(* CoDeSys 2.3.9.59 project: wago_881.pro *)
(* Libraries: WagoLibEthernet_01.lib*10.7.18 06:47:36, SysLibSockets.lib 10.2.11 08:20:54, DALI_02_v2.12.lib*17.1.19 11:19:38, WagoLibReset.lib 2.12.10 13:48:32, SysLibFile.lib 2.12.10 13:48:34, DMXStageProfi_01.lib*19.6.19 09:17:07, Visual.lib 2.12.10 13:48:34, mod_com.lib 2.12.10 13:48:32, Ethernet.lib 2.12.10 13:48:32, SysLibGetAddress.lib 2.12.10 13:48:32, SysLibTime.lib 2.12.10 13:48:32, Standard.lib 2.12.10 13:48:34, SYSLIBCALLBACK.LIB 2.12.10 13:48:32 *)

(* PLC configuration (modules and I/O channels)
K-Bus [K_Bus] node 0, in %IB0 out %QB0
Fieldbus variables [FB_VARS] node 1, in %IB512 out %QB512
*)

(* Task configuration *)
TASK MainTask (PRIORITY := 1); (* freewheeling *)
	PLC_PRG();
END_TASK
TASK DMXTask (PRIORITY := 2, INTERVAL := T#10ms);
	DMX();
END_TASK

(* Global variable list: Variables_Globales *)
VAR_GLOBAL
	ConfigDone: BOOL := FALSE; (* Do the config only one time *)
	info : ARRAY[0..63] OF MODULE_INFO; (* I/O Module infos *)

	LedMode: BYTE := 0;

	(* modules infos *)
	nb_module: BYTE;
	nb_module_in: BYTE;
	nb_module_out: BYTE;
	nb_module_analog_in: BYTE;
	nb_module_analog_out: BYTE;
	start_addr_in: WORD;
	start_addr_out: WORD;
	nb_input_digital: WORD;
	nb_output_digital: WORD;

	(* All inputs events *)
	event: ARRAY[0..512] OF INTER_EVENT; (* See Rules mapping below *)
	lights: ARRAY[0..63] OF BYTE;	(* MAX of 256/8 = 32 digital output modules as lights *)
									(* We store only the boolean state of each light *)
	volets: ARRAY[0..512] OF VOLET; (* MAX of 256/8 = 32 digital output modules as volets *)

	HEARTBEAT: BOOL := FALSE;

	OutArrState: ARRAY[0..512] OF BYTE;	(* state of outputs *)

	impulse_time: TIME := T#300ms;

	(* DALI *)
	DALIJoblist: FbDALI_Joblist;

	Dali_switch: FbDALI_SwitchValue;
	DALIDimmValue: FbDALI_StatusDimmValue;

	(*
		Modbus addresses mapping:
			- [4096..4352] : Standard digital outputs
			- [6144..6244] : KNX inputs/outputs
	*)

	netOutStandard AT %IB512: ARRAY[0..31] OF BYTE;

	netOutKNX AT %IB768: ARRAY[0..12] OF BYTE;
	netInKNX AT %QB768: ARRAY[0..12] OF BYTE;

	write_word: WRITE_OUTPUT_WORD;
	write_bit: WRITE_OUTPUT_BIT;
	read_bit: READ_INPUT_BIT;

END_VAR
VAR_GLOBAL RETAIN
	(* Rules mapping:
		- [0..256] : standard digital inputs
		- [257..357]: knx digital inputs
	*)
	output_type: ARRAY[0..512] OF OUTPUT_TYPE; (* The type of each output *)
	output_addr: ARRAY[0..512] OF OUTPUT_ADDR; (* The addresses for each type *)

    volets_position: ARRAY[0..100] OF DWORD;

	(* DMX Values *)
	abDMX_Values: ARRAY [1..255] OF BYTE;
END_VAR

(* Data type *)
TYPE OUTPUT_ADDR :
STRUCT

	(* the first ouput address, only needed *)
	ADDR1: WORD;
	(* the second address used only for the VOLET function bloc *)
	ADDR2: WORD;

	(* If SameAs <> -1, then a input is wired the same as the specified ID *)
	SameAs: INT := -1;

END_STRUCT
END_TYPE

(* Data type *)
(* Enumerate all type of output.
	NONE: Do nothing.
	TELERUPTEUR: Simulate a telerupteur.
	DIRECT: The input is directly "wired" to the output.
	VOLET: Simulate a volet with one button and 2 output (up and down).
	TELERUPTEUR_DALI: Controls a DALI lamp
	TELERUPTEUR_DALI_GROUP: Controls a DALI group
	KNX_OUTPUT: Simulate a telerupteur with a KNX bool output
*)

TYPE OUTPUT_TYPE : (NONE,
					TELERUPTEUR, DIRECT,
					VOLET, VOLET_IMPULSE,
					TELERUPTEUR_DALI,
					TELERUPTEUR_DALI_GROUP,
					TELERUPTEUR_KNX_OUTPUT,
					DIRECT_KNX_OUTPUT);
END_TYPE

(* Data type *)
TYPE typEthernet_BUFFER :
	STRUCT
		Index		:	INT;
		Data		:	ARRAY[1..1500] OF BYTE;
	END_STRUCT
END_TYPE

(* Data type *)
(* Enumerate all type of output.
	NONE: Do nothing.
	TELERUPTEUR: Simulate a telerupteur.
	DIRECT: The input is directly "wired" to the output.
	VOLET: Simulate a volet with one button and 2 output (up and down).
*)

TYPE VOLET_MODE : (VOLET_STOP, VOLET_UP, VOLET_DOWN, IMP_UP, IMP_DOWN, IMP_STOP);
END_TYPE

(* POU PLC_PRG, ST *)
PROGRAM PLC_PRG
VAR
	i: INT;
	j: INT;
	start: BYTE;
	init_dali: BOOL := FALSE;
	valw: WORD;
	led: LedUsr;
END_VAR
(* Main PRG *)
Config_File_XML();

led(Mode := LedMode);

(* Start the config program *)
Config;

IF (Config.CONFIG_DALI = TRUE) THEN

	(* Call DALI jobs to send commands on the DALI bus *)
	DALIJoblist();
	DALI_Config();

	IF (init_dali = FALSE) THEN
		Dali_switch(xButton := FALSE);
		Dali_switch(bAddress := 255, xGroup := FALSE, bDimmLevel := 0,
				         xButton := TRUE);

		init_dali := TRUE;
	END_IF

END_IF

(* Read inputs and send their status on the network if they changed *)
SendInput;

(* Read a command from UDP *)
UDPServer;

IF (HEARTBEAT = FALSE) THEN
 	ManageOutput;
END_IF

IF (HEARTBEAT = FALSE) THEN

	j := start_addr_out / 8;
	FOR i := start_addr_out / 16 TO 15 DO
		valw := OutArrState[j + 1];
		write_word(WORD_ADDRESS := i, VALUE := SHL(valw, 8) + OutArrState[j]);
		j := j + 2;
	END_FOR
ELSE

	j := 0;
	FOR i := 0 TO 14 DO
		valw := netOutStandard[j + 1];
		write_word(WORD_ADDRESS := i + start_addr_out / 16, VALUE := SHL(valw, 8) + netOutStandard[j]);
		j := j + 2;
		OutArrState[j] := netOutStandard[j];
		OutArrState[j + 1] := netOutStandard[j + 1];
	END_FOR

END_IF
END_PROGRAM

(* POU LedUsr, ST *)
FUNCTION_BLOCK LedUsr
VAR_INPUT
	Mode: BYTE;

END_VAR
VAR_OUTPUT
END_VAR
VAR
	Sequence: ARRAY [0..4] OF FLASHING_SEQUENCE;
	ptrFS: POINTER TO FLASHING_SEQUENCE;

	i: BYTE := 0;
END_VAR
CASE Mode OF
	0 : i := 0;
	1 : i := 11; (* Mode Wago *)
	2 : i := 12; (* Mode PC *)
	3 : i := 13; (* Error *)
END_CASE

LedMode := 255;

CASE i OF
	0 : (* Init *)
		Sequence[0].Colour := ORANGE;
		Sequence[0].Frequency := 10;
		Sequence[0].Relation := 128;
		Sequence[0].Duration := t#0s;

		Sequence[1].Colour := ORANGE;
		Sequence[1].Frequency := 0;
		Sequence[1].Relation := 128;
		Sequence[1].Duration := t#0s;

		Sequence[2].Colour := GREEN;
		Sequence[2].Frequency := 0;
		Sequence[2].Relation := 128;
		Sequence[2].Duration := t#0s;

		Sequence[3].Colour := RED;
		Sequence[3].Frequency := 0;
		Sequence[3].Relation := 128;
		Sequence[3].Duration := t#0s;

		Sequence[4].Colour := ORANGE;
		Sequence[4].Frequency := 0;
		Sequence[4].Relation := 0;
		Sequence[4].Duration := t#0s;

		ptrFS := ADR(Sequence);
		SET_FLASHING_SEQUENCE(TRUE, ADR(ptrFS));

		i := 10;

	10: (* Start *)
		SET_FLASHING_SEQUENCE_INDEX(TRUE, TRUE, 0);
		START_FLASHING_SEQUENCE(TRUE);

		i := 255;

	11: (* Led Mode wago *)
		SET_FLASHING_SEQUENCE_INDEX(TRUE, TRUE, 1);

		i := 255;

	12: (* Led Mode PC *)
		SET_FLASHING_SEQUENCE_INDEX(TRUE, TRUE, 2);

		i := 255;

	13: (* Led Error *)
		SET_FLASHING_SEQUENCE_INDEX(TRUE, TRUE, 3);

		i := 255;

END_CASE
END_FUNCTION_BLOCK

(* POU Config_File_XML, ST *)
PROGRAM Config_File_XML
VAR RETAIN
	wModuleCount : WORD;
END_VAR
VAR CONSTANT
	STRING_1: STRING := '<?xml version="1.0" encoding="ISO-8859-1"?>$r$n';
	STRING_2: STRING := '<?xml-stylesheet type="text/xsl" href="/webserv/cplcfg/EA-config.xsl" ?>$R$n';
	STRING_3: STRING := '<WAGO>$R$n';
	STRING_4: STRING := '<Module ARTIKELNR="" MAP="PLC" LOC="ALL"></Module>$R$n';
	STRING_5: STRING := '</WAGO>$r$n';
END_VAR
VAR
	info : ARRAY[0..63] OF MODULE_INFO;
	access: MODULE_INFO_ACCESS;
	i: INT := 0;
	Status: BYTE := 0;
	DetectedModules: INT;
	FileHandle: DWORD;
	dwWrite: DWORD;
	NumberOfEntries: BYTE := 0;
	FileIsClosed: BOOL;
END_VAR
CASE Status OF
	0 :	ADD_PI_INFORMATION(EN:=TRUE, pAccess:=ADR(access), pInfo:=ADR(info));
		i:=0;
		WHILE info[i].physicalPos<>0
			DO
			i:=i+1;
		END_WHILE
		DetectedModules := i;
		Status := Status +1;
	1 :	IF DetectedModules = wModuleCount
			THEN
			Status := 255; (* Done *)
		ELSE
			Status := 10;
		END_IF
	10:	FileHandle:=SysFileOpen(FileName:='\etc\EA-config.xml', Mode:='w');
		IF FileHandle <> 0 THEN
			Status := Status+1;
		END_IF
	11:	dwWrite:=SysFileWrite(File:=FileHandle, Buffer:=ADR(STRING_1), Size:=LEN(STRING_1));
		IF dwWrite=LEN(STRING_1) THEN
			Status := Status+1;
		END_IF
	12:	dwWrite:=SysFileWrite(File:=FileHandle, Buffer:=ADR(STRING_2), Size:=LEN(STRING_2));
		IF dwWrite=LEN(STRING_2) THEN
			Status := Status+1;
		END_IF
	13:	dwWrite:=SysFileWrite(File:=FileHandle, Buffer:=ADR(STRING_3), Size:=LEN(STRING_3));
		IF dwWrite=LEN(STRING_3) THEN
			Status := Status+1;
		END_IF
	14:	dwWrite:=SysFileWrite(File:=FileHandle, Buffer:=ADR(STRING_4), Size:=LEN(STRING_4));
		IF dwWrite=LEN(STRING_4) THEN
			Status := Status+1;
			NumberOfEntries := NumberOfEntries+1;
		END_IF
	15: IF NumberOfEntries < DetectedModules
			THEN
			Status := Status -1;
		ELSE
			Status := Status +1;
		END_IF
	16:	dwWrite:=SysFileWrite(File:=FileHandle, Buffer:=ADR(STRING_5), Size:=LEN(STRING_5));
		IF dwWrite=LEN(STRING_5) THEN
			Status := Status+1;
		END_IF
	17:	FileIsClosed := SysFileClose(File:= FileHandle);
		IF FileIsClosed
			THEN
			Status := 20;
		END_IF
	20:	wModuleCount := DetectedModules;
		FirmwareReset(EN := TRUE);
END_CASE
END_PROGRAM

(* POU Config, ST *)
PROGRAM Config
VAR
	access : MODULE_INFO_ACCESS;
	cpt: BYTE;
	ethernet_config : ETHERNET_SET_VARIABLES;
	CONFIG_DALI: BOOL;
	first_in: BOOL := FALSE;
	first_out: BOOL := FALSE;
END_VAR
VAR_INPUT RETAIN
	SERVER_IP: DWORD;
	DALI_MODE: BYTE;
END_VAR
VAR CONSTANT
	CALAOS_VERSION_H: WORD := 2;
	CALAOS_VERSION_L: WORD := 3;
	DALI: BYTE := 1;
	DSI: BYTE := 2;
END_VAR
(* Do all the config job *)

IF (ConfigDone = FALSE) THEN

(* Get the module I/O Config *)
access.physicalPosTo := 0;
access.moduleType := 0;
ADD_PI_INFORMATION( 1, ADR(access), ADR(info[0]) );

FOR cpt := 0 TO 63 DO
	IF (info[cpt].moduleType = 0 AND info[cpt].physicalPos = 0) THEN
		cpt := 63; (* the end *)
	ELSE
		IF (info[cpt].moduleType = 641) THEN
			(* This is a DALI module *)
			CONFIG_DALI := TRUE;
		END_IF

		nb_module := nb_module + 1;
		IF ((info[cpt].desc.sizePAE > 8) AND (info[cpt].desc.channels > 0)) THEN
			nb_module_analog_in := nb_module_analog_in + 1;
(*			start_addr_in := start_addr_in + info[cpt].desc.sizePAE; *)
		END_IF
		IF ((info[cpt].desc.sizePAA > 8) AND (info[cpt].desc.channels > 0)) THEN
			nb_module_analog_out := nb_module_analog_out + 1;
(*			start_addr_out := start_addr_out + info[cpt].desc.sizePAA; *)
		END_IF
		IF ((info[cpt].desc.sizePAE <= 16) AND (info[cpt].desc.sizePAE > 0) AND (info[cpt].desc.channels = 0)) THEN
			nb_module_in := nb_module_in + 1;
			nb_input_digital := nb_input_digital + info[cpt].desc.sizePAE;

			IF (first_in = FALSE) THEN
				first_in := TRUE;
				start_addr_in := info[cpt].desc.posPAE;
			END_IF
		END_IF
		IF ((info[cpt].desc.sizePAA <= 16) AND (info[cpt].desc.sizePAA > 0) AND (info[cpt].desc.channels = 0)) THEN
			nb_module_out := nb_module_out + 1;
			nb_output_digital := nb_output_digital + info[cpt].desc.sizePAA;

			IF (first_out = FALSE) THEN
				first_out := TRUE;
				start_addr_out := info[cpt].desc.posPAA;
			END_IF
		END_IF

	END_IF
END_FOR

(* Start the heartbeat timer *)
(*HEARTBEAT_TIMER(IN:=FALSE, PT:=T#30s);*)
(*HEARTBEAT_TIMER(IN:=TRUE, PT:=T#30s);*)

(* Config du timout des sockets *)
ethernet_config(EN:=TRUE, BootpRequest:=0, ConnectionWdTime:=65535);

ConfigDone := TRUE;

END_IF
END_PROGRAM

(* POU SendInput, ST *)
PROGRAM SendInput
VAR
	cpt: INT;

	eth: Ethernet_Client;
	wBuffer: POINTER TO BYTE;
	command: STRING(255);
	start_send: BOOL := FALSE;
	ReceiveData: typEthernet_buffer;
	Write: ETHERNET_WRITE_PT;
	socket:	WORD;
END_VAR
(* Get all inputs *)

(* Get the address of the first digital input *)
FOR cpt := 0 TO UINT_TO_BYTE(nb_input_digital) DO
	event[cpt](IN := GetInput(cpt + start_addr_in));

	(* Send inputs to network *)
	IF (event[cpt].ON = TRUE) THEN
		command := 'WAGO INT ';
		command := CONCAT(command,  INT_TO_STRING(cpt));
		command := CONCAT(command,  ' 1');

		Write(EN := 0, SOCKET := 0, LEN_IN := 0, DST_IP:=0, DST_PORT:=0, DATA_PT := wBuffer);
		Write(EN := 1, SOCKET := socket, LEN_IN := LEN(command), DST_IP := Config.SERVER_IP, DST_PORT := 4646, DATA_PT := wBuffer);
	END_IF
	IF (event[cpt].OFF = TRUE) THEN
		command := 'WAGO INT ';
		command := CONCAT(command,  INT_TO_STRING(cpt));
		command := CONCAT(command,  ' 0');

		Write(EN := 0, SOCKET := 0, LEN_IN := 0, DST_IP:=0, DST_PORT:=0, DATA_PT := wBuffer);
		Write(EN := 1, SOCKET := socket, LEN_IN := LEN(command), DST_IP := Config.SERVER_IP, DST_PORT := 4646, DATA_PT := wBuffer);
	END_IF
END_FOR

wBuffer := ADR(command);

eth(xOPEN_CLIENT := TRUE, wIP := Config.SERVER_IP, wPort := 4646,
	xTCP_PROTOCOL := FALSE, iBYTES_TO_SEND := LEN(command) + 1,
	ptSEND_BUFFER := wBuffer, xSTART_SEND := start_send,
	utRECEIVE_BUFFER := ReceiveData);

socket := eth.MyEthernetOpen.SOCKET;
END_PROGRAM

(* POU Ethernet_Client, ST *)
FUNCTION_BLOCK Ethernet_Client
(************************************************************)
(* ETHERNET_CLIENT		                             			*)
(* Ver. 1.0                                      			          			*)
(* Date    :  10.02.2003					          			*)
(* Author :  Volker Begemann                                       		*)
(************************************************************)
VAR_INPUT
	xOPEN_CLIENT			:	BOOL;			(* Set TRUE to enable function block			*)
	wIP						:	DWORD;		(* IP Address of server						*)
	wPORT					:	WORD;		(* Port number								*)
	xTCP_PROTOCOL		:	BOOL;			(* TRUE => TCP; FALSE => UDP				*)
	iBYTES_TO_SEND		:	INT;			(* Number of bytes to transmit				*)
	ptSEND_BUFFER			:	POINTER TO ARRAY[1..1500] OF BYTE;	(* Transmit Buffer	*)
END_VAR
VAR_IN_OUT
	xSTART_SEND			:	BOOL;			(* Set TRUE to initiate data transmittal, will be	*)
													(* reset FALSE when transmittal is completed 	*)
	utRECEIVE_BUFFER		:	typEthernet_BUFFER;	(* Receive Buffer *)
END_VAR
VAR_OUTPUT
	utERROR					:	ETH_ERROR;	(* See ETH_ERROR datatype in ETHERNET.LIB	*)
													(* for error codes and definitions						*)
	xCLIENT_OPEN			:	BOOL;			(* TRUE if socket connection made					*)
	wSOCKET					:	WORD;		(* Socket connection number							*)
END_VAR
VAR
	MyEthernetOpen				: ETHERNET_CLIENT_OPEN;
	MyEthernetClose				: ETHERNET_CLIENT_CLOSE;
	MyEthernetWrite				: ETHERNET_WRITE;
	MyEthernetRead				: ETHERNET_READ;
	EthernetBuffer					: ARRAY[1..1500] OF BYTE;
	Status							: WORD:=0;
	i								: INT;
	GetConfig						: ETHERNET_GET_NETWORK_CONFIG;
	Protocol						: WORD;
	ProtocolType					: WORD;
	CloseState						:INT;
END_VAR
IF xOpen_Client THEN

	CASE Status OF
		0:(*Initialize functionblocks*)
			GetConfig(EN:=FALSE );
			GetConfig(EN:=TRUE );
			status:=1;
			utERROR:=0;
			wSocket:=0;
			closeState:=0;
			xCLIENT_OPEN:=FALSE;

			IF xTCP_PROTOCOL THEN
				Protocol		:= IPPROTO_TCP; (*TCP*)
				ProtocolType	:= SOCK_STREAM;
			ELSE
				Protocol		:= IPPROTO_UDP;(*UDP*)
				ProtocolType	:= SOCK_DGRAM;
			END_IF

		1:(*check ethernet stack*)
			GetConfig(EN:=TRUE );
			IF GetConfig.ENO THEN
				IF GetConfig.IP_ADR<>0 THEN
					status:=4;(*stack initialized*)
				ELSE
					status:=0;(*try again*)
				END_IF
			END_IF

	
		4:(*open connection*)
			MyEthernetRead(	EN:= 0, SOCKET:=0 ,  DATA:=EthernetBuffer );
			MyEthernetClose(EN:= 0);
			MyEthernetOpen(EN:=0);

			MyEthernetOpen(EN:=1 , TYP:=ProtocolType	 , PROTO:=Protocol , IP_ADR:= wIP, PORT:=wPort );

			status:=5;

		5:(*wait for server response according to client  request to open the connection*)
			MyEthernetOpen(EN:=1, TYP:=ProtocolType, PROTO:=Protocol, IP_ADR:= wIP, PORT:=wPort );
			IF  MyEthernetOpen.ENO = 1 THEN
				IF MyEthernetOpen.ERROR = 0 THEN
					Status  := 10; (*socket available*)
					xCLIENT_OPEN:=TRUE;
					wSOCKET	:=MyEthernetOpen.socket;
				ELSE
					Status := 0; (*no socket available, try it again *)
				END_IF;
				utERROR:=MyEthernetOpen.ERROR;
			END_IF


		10:(* Monitor ethernet port for new data *)

	 		MyEthernetRead(	EN:= 1, SOCKET:=MyEthernetOpen.SOCKET ,  DATA:=EthernetBuffer );
			MyEthernetRead(	EN:= 0, SOCKET:=0 ,  DATA:=EthernetBuffer );

			utERROR:=MyEthernetREAD.ERROR;
			IF(MyEthernetRead.ERROR<>0) THEN  (* Error reading the socket, close it *)
				Status:=40;
			ELSIF (MyEthernetRead.LEN_OUT <>0) THEN  (* Process the data received via the ethernet port *)
				Status:=20;
				ELSIF (iBytes_TO_SEND > 0 AND xSTART_SEND) THEN  (* Process the data put in the send_buffer *)
				status:=30;
				MyEthernetWrite(	EN:= 0 , DATA:=EthernetBuffer );
			END_IF

		20:	(* Copy the data received via the ethernet port to the receive buffer*)

			FOR i := 1 TO MyEthernetRead.LEN_OUT DO
				utReceive_buffer.index :=(utReceive_buffer.index MOD 1500)+1;
				utReceive_buffer.data[utReceive_buffer.index] := EthernetBuffer[i];
			END_FOR
			Status:=10;

		30: (* Process the data in the send buffer *)

			EthernetBuffer :=ptSEND_BUFFER^;
			MyEthernetWrite(	EN:= 1,SOCKET:= MyEthernetOpen.SOCKET,
								LEN_IN:=iBYTES_TO_SEND,DATA:=EthernetBuffer );

			IF MyEthernetWrite.eno THEN
				IF(MyEthernetWrite.ERROR <>0) THEN
					Status:=40;(* Error writing to the socket, close it *)
				ELSE
					Status:=10; (* Comms complete, read more data *)
				END_IF;
				xSTART_SEND:=FALSE;
				utERROR:=MyEthernetWrite.ERROR;
			END_IF

		40:	(* Close the client *)

			MyEthernetClose(EN:= 1, SOCKET:= MyEthernetOpen.SOCKET);
			IF MyEthernetClose.eno THEN
				MyEthernetClose(EN:= 0);
				xCLIENT_OPEN:=FALSE;
				Status := 0; (* Try to open the server again *)
			END_IF
	
	END_CASE;
ELSE
	CASE CloseState OF
	0:
		MyEthernetClose(EN:= 0);
		MyEthernetClose(EN:= 1, SOCKET:= MyEthernetOpen.SOCKET);
		CloseState:=1;
	1:
		MyEthernetClose(EN:= 1, SOCKET:= MyEthernetOpen.SOCKET);
		IF MyEthernetClose.eno THEN
			MyEthernetClose(EN:= 0);
			CloseState:=2;
		END_IF
	2:
		Status := 0;
		utERROR:=0;
		xCLIENT_OPEN:=FALSE;
	END_CASE
END_IF
END_FUNCTION_BLOCK

(* POU GetInput, ST *)
FUNCTION GetInput : BOOL
VAR_INPUT
	bit_offset: UINT;
END_VAR
VAR
END_VAR
VAR CONSTANT
	byBitArr: ARRAY[0..7] OF BYTE := 16#01,16#02,16#04,16#08,16#10,16#20,16#40,16#80;
END_VAR
(* get the byte AND  select the bit *)

read_bit(WORD_ADDRESS := bit_offset / 16, BIT_ADDRESS := bit_offset MOD 16);

GetInput := read_bit.VALUE;
END_FUNCTION

(* POU UDPServer, ST *)
PROGRAM UDPServer
VAR
	server: EthernetServer_FB;

	rBuffer, wBuffer: POINTER TO BYTE;
	buffer: ARRAY[1 .. 1500] OF BYTE;
	cmd: STRING(255);
	start_send: BOOL := FALSE;
	i: WORD;
	dali_group: BOOL;

	HEARTBEAT_TIMER: TON;

	p1: DINT;
	p2: DINT;
	p3: DINT;
	p4: DINT;
	p5: DINT;
	p6: DINT;
	p7: DINT;
	p8: DINT;
	ip1, ip2, ip3, ip4: DWORD;
	DaliSend: BOOL := FALSE;

	(* Used by dali config for answer
	   0 = no action
	   1 = Search all active address
	   2 = Read groups for short adress
	   3 = Switch on/off all lamps
	  98 = Addresing query
	  99 = Addressing in progress
	*)
	DaliSendAction: BYTE := 0;

	(* Dali config FB *)
	DALIShowShortAdr: FbDALI_ShowShortAdr;
	DALIConfigDevice: FbDALI_ConfigDevice;
	DALIConfigShortAddress: FbDALI_ConfigShortAddress;
	DALIMaster: FbDALI_Master;
	DALIMasterAdv: FbDALI_Master_Adv;

	extendedAddr: BOOL;
	newAddressing: BOOL;
	resetAddr: BOOL;
	replaceAddr: BOOL;
	delAddressing: BOOL;
	oldAddr, newAddr, delAddr: BYTE;
	dali_master: BOOL;
	group_address: BYTE;
	groups_cmd_1_8: BYTE;
	addr_1_16: WORD;
	addr_17_32: WORD;

	dmx_read_addr: BYTE;

END_VAR
(* Here we start an UDP server for other network functions *)

HEARTBEAT_TIMER(IN:=TRUE, PT:=T#30s);

rBuffer := ADR(buffer);
wBuffer := ADR(cmd);

(* cmd := CONCAT(cmd, ASCIIBYTE_TO_STRING(0)); *)

server.tTIMEOUT	:= t#60s;
server.xTCP_PROTOCOL := FALSE;
server.wPORT := 4646;
server.iBYTES_TO_SEND := LEN(cmd) + 1;
server(xOPEN_SERVER := TRUE, xSTART_SEND := start_send, ptSEND_BUFFER := wBuffer, ptRECV_BUFFER := rBuffer);

IF server.bDataReceived THEN

	cmd := '';
	FOR i := 1 TO server.iBYTES_RECEIVED DO
		cmd := CONCAT(cmd, ASCIIBYTE_TO_STRING(buffer[i]));
	END_FOR

	IF (STRING_COMPARE(cmd, 'WAGO_HEARTBEAT') = TRUE) THEN
		HEARTBEAT_TIMER(IN:=FALSE, PT:=T#30s);
		HEARTBEAT_TIMER(IN:=TRUE, PT:=T#30s);

		LedMode := 2;
	END_IF

	IF (Strncmp(cmd, 'WAGO_SET_OUTTYPE ', 17) = TRUE) THEN
		p1 := GET_PARAM_DINT(cmd, 1);
		p2 := GET_PARAM_DINT(cmd, 2);
		CASE p2 OF
		0: output_type[p1] := NONE;
		1: output_type[p1] := TELERUPTEUR;
		2: output_type[p1] := DIRECT;
		3: output_type[p1] := VOLET;
		4: output_type[p1] := VOLET_IMPULSE;
		5: output_type[p1] := TELERUPTEUR_DALI;
		6: output_type[p1] := TELERUPTEUR_DALI_GROUP;
		7: output_type[p1] := TELERUPTEUR_KNX_OUTPUT;
		8: output_type[p1] := DIRECT_KNX_OUTPUT;
		END_CASE
	END_IF

	IF (Strncmp(cmd, 'WAGO_SET_OUTADDR ', 17) = TRUE) THEN
		p1 := GET_PARAM_DINT(cmd, 1);
		p2 := GET_PARAM_DINT(cmd, 2);
		p3 := GET_PARAM_DINT(cmd, 3);
		p4 := GET_PARAM_DINT(cmd, 4);
		output_addr[p1].ADDR1 := DINT_TO_BYTE(p2);
		output_addr[p1].ADDR2 := DINT_TO_BYTE(p3);
		output_addr[p1].SameAs := DINT_TO_INT(p4);
	END_IF

	IF (Strncmp(cmd, 'WAGO_GET_OUTTYPE ', 17) = TRUE) THEN
		p1 := GET_PARAM_DINT(cmd, 1);
		cmd := 'WAGO_OUTTYPE ';
		cmd := CONCAT(cmd, ITOA(DINT_TO_INT(p1)));
		cmd := CONCAT(cmd, ' ');
		CASE output_type[p1] OF
		NONE: cmd := CONCAT(cmd, ITOA(0));;
		TELERUPTEUR: cmd := CONCAT(cmd, ITOA(1));;
		DIRECT: cmd := CONCAT(cmd, ITOA(2));;
		VOLET: cmd := CONCAT(cmd, ITOA(3));;
		VOLET_IMPULSE: cmd := CONCAT(cmd, ITOA(4));;
		TELERUPTEUR_DALI: cmd := CONCAT(cmd, ITOA(5));;
		TELERUPTEUR_DALI_GROUP: cmd := CONCAT(cmd, ITOA(6));;
		TELERUPTEUR_KNX_OUTPUT: cmd := CONCAT(cmd, ITOA(7));;
		DIRECT_KNX_OUTPUT: cmd := CONCAT(cmd, ITOA(8));;
		END_CASE
		start_send := TRUE;
	END_IF

	IF (Strncmp(cmd, 'WAGO_GET_OUTADDR ', 17) = TRUE) THEN
		p1 := GET_PARAM_DINT(cmd, 1);
		cmd := 'WAGO_OUTADDR ';
		cmd := CONCAT(cmd, ITOA(DINT_TO_INT(p1)));
		cmd := CONCAT(cmd, ' ');
		cmd := CONCAT(cmd, ITOA(output_addr[p1].ADDR1));
		cmd := CONCAT(cmd, ' ');
		cmd := CONCAT(cmd, ITOA(output_addr[p1].ADDR2));
		cmd := CONCAT(cmd, ' ');
		cmd := CONCAT(cmd, ITOA(output_addr[p1].SameAs));
		start_send := TRUE;
	END_IF

	IF (STRING_COMPARE(cmd, 'WAGO_GET_INFO') = TRUE) THEN
		cmd := 'WAGO_INFO ';
		cmd := CONCAT(cmd, ITOA(nb_module));
		cmd := CONCAT(cmd, ' ');
		cmd := CONCAT(cmd, ITOA(nb_module_in));
		cmd := CONCAT(cmd, ' ');
		cmd := CONCAT(cmd, ITOA(WORD_TO_INT(nb_module_out)));
		cmd := CONCAT(cmd, ' ');
		cmd := CONCAT(cmd, ITOA(WORD_TO_INT(nb_input_digital)));
		cmd := CONCAT(cmd, ' ');
		cmd := CONCAT(cmd, ITOA(WORD_TO_INT(nb_output_digital)));
		cmd := CONCAT(cmd, ' ');
		cmd := CONCAT(cmd, ITOA(nb_module_analog_in));
		cmd := CONCAT(cmd, ' ');
		cmd := CONCAT(cmd, ITOA(nb_module_analog_out));
		start_send := TRUE;
	END_IF

	IF (Strncmp(cmd, 'WAGO_GET_INFO_MODULE ', 21) = TRUE) THEN
		p1 := GET_PARAM_DINT(cmd, 1);
		cmd := 'WAGO_MODULE ';
		cmd := CONCAT(cmd, ITOA(DINT_TO_INT(p1)));
		cmd := CONCAT(cmd, ' ');
		cmd := CONCAT(cmd, ITOA(WORD_TO_INT(info[p1].moduleType)));
		cmd := CONCAT(cmd, ' ');
		cmd := CONCAT(cmd, ITOA(info[p1].physicalPos));
		cmd := CONCAT(cmd, ' ');
		cmd := CONCAT(cmd, ITOA(info[p1].desc.sizePAE));
		cmd := CONCAT(cmd, ' ');
		cmd := CONCAT(cmd, ITOA(info[p1].desc.sizePAA));
		start_send := TRUE;
	END_IF

	IF (Strncmp(cmd, 'WAGO_SET_SERVER_IP ', 19) = TRUE) THEN
		cmd := DELETE(cmd, 19, 1);
		(* deletes the dot  *)
		cmd := REPLACE(cmd, ' ', 1, FIND(cmd, '.'));
		cmd := REPLACE(cmd, ' ', 1, FIND(cmd, '.'));
		cmd := REPLACE(cmd, ' ', 1, FIND(cmd, '.'));
		ip1 := GET_PARAM_DINT(cmd, 0);
		ip2 := GET_PARAM_DINT(cmd, 1);
		ip3 := GET_PARAM_DINT(cmd, 2);
		ip4 := GET_PARAM_DINT(cmd, 3);
		Config.SERVER_IP := SHL(ip1, 24) OR SHL(ip2, 16) OR SHL(ip3, 8) OR ip4;
	END_IF


	IF (Strncmp(cmd, 'WAGO_SET_DMX_IP ', 16) = TRUE) THEN
		cmd := DELETE(cmd, 16, 1);
		DMX.IPaddress := cmd;
	END_IF

	IF (Strncmp(cmd, 'WAGO_SET_OUTPUT ', 16) = TRUE) THEN
		p1 := GET_PARAM_DINT(cmd, 1);
		p2 := GET_PARAM_DINT(cmd, 2);

		p1 := start_addr_out + p1;

		IF (p2 = 1) THEN
			SetOutput(DINT_TO_UINT(p1), TRUE);
		ELSE
			SetOutput(DINT_TO_UINT(p1), FALSE);
		END_IF
	END_IF

	IF (Strncmp(cmd, 'WAGO_GET_VERSION', 16) = TRUE) THEN
		cmd := 'WAGO_GET_VERSION ';
		cmd := CONCAT(cmd, ITOA(WORD_TO_INT(Config.CALAOS_VERSION_H)));
		cmd := CONCAT(cmd, '.');
		cmd := CONCAT(cmd, ITOA(WORD_TO_INT(Config.CALAOS_VERSION_L)));
		cmd := CONCAT(cmd, ' 750-841');
		start_send := TRUE;
	END_IF

	IF (Strncmp(cmd, 'WAGO_DALI_SET ', 14) = TRUE AND DaliSendAction = 0) THEN
		p1 := GET_PARAM_DINT(cmd, 1); (* Dali Line *)
		p2 := GET_PARAM_DINT(cmd, 2); (* Short addr or group? *)
		p3 := GET_PARAM_DINT(cmd, 3); (* Dali Address *)
		p4 := GET_PARAM_DINT(cmd, 4); (* Dimm value in percent *)
		p5 := GET_PARAM_DINT(cmd, 5); (* Fade time *)

		IF (p2 = 1) THEN
			dali_group := TRUE;
		ELSE
			dali_group := FALSE;
		END_IF

		IF (p3 > 99) THEN
			abDMX_Values[DINT_TO_BYTE(p3 - 100)] := DINT_TO_BYTE(p4 * 255 / 100);
		ELSE
			Dali_switch(xButton := FALSE);
			Dali_switch(bAddress := DINT_TO_BYTE(p3), xGroup := dali_group, bDimmLevel := DINT_TO_BYTE(p4),
				bFadeTime := DINT_TO_BYTE(p5), xButton := TRUE);
		END_IF
	END_IF

	IF (Strncmp(cmd, 'WAGO_DALI_GET ', 14) = TRUE AND DaliSendAction = 0) THEN
		p1 := GET_PARAM_DINT(cmd, 1); (* Dali Line *)
		p2 := GET_PARAM_DINT(cmd, 2); (* Short addr *)
		p3 := GET_PARAM_DINT(cmd, 3); (* Dali Address *)
		p4 := GET_PARAM_DINT(cmd, 4); (* Dimm value in percent *)
		p5 := GET_PARAM_DINT(cmd, 5); (* Fade time *)

		IF (p2 = 1) THEN
			dali_group := TRUE;
		ELSE
			dali_group := FALSE;
		END_IF

		IF (p3 < 99) THEN
			DALIDimmValue(xEnable := TRUE, bShortAddress := DINT_TO_BYTE(p2), tCycleTime := t#1s);
			dmx_read_addr := 0;
		ELSE
			dmx_read_addr := DINT_TO_BYTE(p3 - 100);
		END_IF
		DaliSend := TRUE;
	END_IF

    IF (Strncmp(cmd, 'WAGO_INFO_VOLET_GET ', 20) = TRUE) THEN
		p1 := GET_PARAM_DINT(cmd, 1);
		cmd := 'WAGO_INFO_VOLET ';
		cmd := CONCAT(cmd, ITOA(DINT_TO_INT(p1)));
		cmd := CONCAT(cmd, ' ');
		cmd := CONCAT(cmd, DWORD_TO_STRING(volets_position[p1]));
		start_send := TRUE;
	END_IF

    IF (Strncmp(cmd, 'WAGO_INFO_VOLET_SET ', 20) = TRUE) THEN
		p1 := GET_PARAM_DINT(cmd, 1);
		p2 := GET_PARAM_DINT(cmd, 2);
		volets_position[p1] := DINT_TO_DWORD(p2);
	END_IF

(*    IF (Strncmp(cmd, 'WAGO_DALI_GET_ADDR', 18) = TRUE) THEN
		DALIShowShortAdr(xQuery := FALSE);
		DALIShowShortAdr(xQuery := TRUE);
		DaliSendAction := 1;
	END_IF *)

	IF (Strncmp(cmd, 'WAGO_DALI_GET_ADDR ', 18) = TRUE) THEN
		p1 := GET_PARAM_DINT(cmd, 1);
		dali_master := TRUE;
		DALIMasterAdv(xStartDaliMaster := dali_master, iCommand := 506);
		DaliSendAction := 1;
	END_IF

	IF (Strncmp(cmd, 'WAGO_DALI_GET_DEVICE_INFO ', 26) = TRUE) THEN
		p1 := GET_PARAM_DINT(cmd, 1);
		p2 := GET_PARAM_DINT(cmd, 2);
		DALIConfigDevice(xQuery := FALSE);
		DALIConfigDevice(xQuery := TRUE, bAddress := DINT_TO_BYTE(p2));
		DaliSendAction := 2;
	END_IF

	IF (Strncmp(cmd, 'WAGO_DALI_GET_DEVICE_GROUP ', 27) = TRUE) THEN
		p1 := GET_PARAM_DINT(cmd, 1);
		p2 := GET_PARAM_DINT(cmd, 2); (* address *)
		group_address := DINT_TO_BYTE(p2);
		dali_master := TRUE;
		DALIMaster(xStartDaliMaster := dali_master, iCommand := 192, bAddress := group_address);
		DaliSendAction := 3;
	END_IF

	IF (Strncmp(cmd, 'WAGO_DALI_DEVICE_ADD_GROUP ', 27) = TRUE) THEN
		p1 := GET_PARAM_DINT(cmd, 1);
		p2 := GET_PARAM_DINT(cmd, 2); (* device address *)
		p3 := GET_PARAM_DINT(cmd, 3); (* group *)
		dali_master := TRUE;
		DALIMasterAdv(xStartDaliMaster := dali_master, iCommand := 501, bCommandValue1 := 95 + DINT_TO_BYTE(p3), bAddress := DINT_TO_BYTE(p2));
		DaliSendAction := 5;
	END_IF

	IF (Strncmp(cmd, 'WAGO_DALI_DEVICE_DEL_GROUP ', 27) = TRUE) THEN
		p1 := GET_PARAM_DINT(cmd, 1);
		p2 := GET_PARAM_DINT(cmd, 2); (* device address *)
		p3 := GET_PARAM_DINT(cmd, 3); (* group *)
		dali_master := TRUE;
		DALIMasterAdv(xStartDaliMaster := dali_master, iCommand := 501, bCommandValue1 := 111 + DINT_TO_BYTE(p3), bAddress := DINT_TO_BYTE(p2));
		DaliSendAction := 6;
	END_IF

	IF (Strncmp(cmd, 'WAGO_DALI_CENTRAL ', 18) = TRUE) THEN
		p1 := GET_PARAM_DINT(cmd, 1);
		p2 := GET_PARAM_DINT(cmd, 2);
		DALIShowShortAdr(xCentr_ON := FALSE, xCentr_OFF := FALSE);
		IF (p2 = 1) THEN
			DALIShowShortAdr(xCentr_ON := TRUE);
		ELSE
			DALIShowShortAdr(xCentr_OFF := TRUE);
		END_IF
	END_IF

	IF (Strncmp(cmd, 'WAGO_DALI_BLINK ', 16) = TRUE) THEN
		p1 := GET_PARAM_DINT(cmd, 1);
		p2 := GET_PARAM_DINT(cmd, 2); (* address *)
		p3 := GET_PARAM_DINT(cmd, 3); (* group? *)
		p4 := GET_PARAM_DINT(cmd, 4); (* blink time *)
		DALIShowShortAdr(xBlink := FALSE);
		DALIShowShortAdr(xBlink := TRUE, bAddress := DINT_TO_BYTE(p2), bBlinkTime := DINT_TO_BYTE(p4), xGroup := DINT_TO_BOOL(p3));
	END_IF

	IF (Strncmp(cmd, 'WAGO_DALI_BLINK_STOP ', 21) = TRUE) THEN
		p1 := GET_PARAM_DINT(cmd, 1);
		DALIShowShortAdr(xBlink_OFF := FALSE);
		DALIShowShortAdr(xBlink_OFF := TRUE);
	END_IF

	IF (Strncmp(cmd, 'WAGO_DALI_SET_DEVICE_CONFIG ', 28) = TRUE) THEN
		p1 := GET_PARAM_DINT(cmd, 1);
		p2 := GET_PARAM_DINT(cmd, 2); (* device address *)
		p3 := GET_PARAM_DINT(cmd, 3); (* fade rate *)
		p4 := GET_PARAM_DINT(cmd, 4); (* fade time *)
		p5 := GET_PARAM_DINT(cmd, 5); (* max level *)
		p6 := GET_PARAM_DINT(cmd, 6); (* min level *)
		p7 := GET_PARAM_DINT(cmd, 7); (* system failure level *)
		p8 := GET_PARAM_DINT(cmd, 8); (* power on level *)
		DALIConfigDevice(xSetConfig := FALSE);
		DALIConfigDevice(xSetConfig := TRUE, bAddress := DINT_TO_BYTE(p2),
					bFade_Rate := DINT_TO_BYTE(p3), bFade_Time := DINT_TO_BYTE(p4),
					bMax_Level := DINT_TO_BYTE(p5), bMin_Level := DINT_TO_BYTE(p6),
					bSystem_Failure_Level := DINT_TO_BYTE(p7), bPower_On_Level := DINT_TO_BYTE(p8));
	END_IF

	IF (Strncmp(cmd, 'WAGO_DALI_ADDRESSING_NEW ', 25) = TRUE) THEN
		p1 := GET_PARAM_DINT(cmd, 1);
		p2 := GET_PARAM_DINT(cmd, 2); (* reset? *)
		DALIConfigShortAddress(xNewAddressing := FALSE);
		DALIConfigShortAddress(xNewAddressing := TRUE, xReset := DINT_TO_BOOL(p2), xSwitchAtAddressing := TRUE);
		DALIConfigShortAddress(xNewAddressing := FALSE); (* double click *)
		DALIConfigShortAddress(xNewAddressing := TRUE, xReset := DINT_TO_BOOL(p2), xSwitchAtAddressing := TRUE);
		replaceAddr := FALSE;
		extendedAddr := FALSE;
		newAddressing := TRUE;
		delAddressing := FALSE;
		resetAddr := DINT_TO_BOOL(p2);
		DaliSendAction := 99; (* addressing in progress *)
	END_IF

	IF (Strncmp(cmd, 'WAGO_DALI_ADDRESSING_ADD ', 25) = TRUE) THEN
		p1 := GET_PARAM_DINT(cmd, 1);
		DALIConfigShortAddress(xExtendedAddressing := FALSE);
		DALIConfigShortAddress(xExtendedAddressing := TRUE, xSwitchAtAddressing := TRUE);
		replaceAddr := FALSE;
		extendedAddr := TRUE;
		newAddressing := FALSE;
		resetAddr := FALSE;
		delAddressing := FALSE;
		DaliSendAction := 99; (* addressing in progress *)
	END_IF

	IF (Strncmp(cmd, 'WAGO_DALI_ADDRESSING_STATUS ', 28) = TRUE) THEN
		p1 := GET_PARAM_DINT(cmd, 1);
		DaliSendAction := 98; (* addressing in progress *)
	END_IF

	IF (Strncmp(cmd, 'WAGO_DALI_ADDRESSING_CHANGE ', 28) = TRUE) THEN
		p1 := GET_PARAM_DINT(cmd, 1);
		p2 := GET_PARAM_DINT(cmd, 2); (* old address *)
		p3 := GET_PARAM_DINT(cmd, 3); (* new address *)
		oldAddr := DINT_TO_BYTE(p2);
		newAddr := DINT_TO_BYTE(p3);
		DALIConfigShortAddress(xReplaceShortAddress := FALSE);
		DALIConfigShortAddress(xReplaceShortAddress := TRUE, bOldShortAddress := oldAddr, bNewShortAddress := newAddr);
		replaceAddr := TRUE;
		extendedAddr := FALSE;
		newAddressing := FALSE;
		resetAddr := FALSE;
		delAddressing := FALSE;
		DaliSendAction := 99; (* addressing in progress *)
	END_IF

	IF (Strncmp(cmd, 'WAGO_DALI_ADDRESSING_DEL ', 25) = TRUE) THEN
		p1 := GET_PARAM_DINT(cmd, 1);
		p2 := GET_PARAM_DINT(cmd, 2); (* address to delete *)
		delAddr := DINT_TO_BYTE(p2);
		DALIConfigShortAddress(xDeleteShortAddress := FALSE);
		DALIConfigShortAddress(xDeleteShortAddress := TRUE, bDeleteShortAddress := delAddr);
		replaceAddr := TRUE;
		extendedAddr := FALSE;
		newAddressing := FALSE;
		resetAddr := FALSE;
		delAddressing := TRUE;
		DaliSendAction := 99; (* addressing in progress *)
	END_IF

END_IF

CASE DaliSendAction OF
(*
1: (* WAGO_DALI_GET_ADDR *)
	IF (DALIShowShortAdr.xReady = TRUE) THEN
		cmd := 'WAGO_DALI_GET_ADDR ';
		cmd := CONCAT(cmd, WORD_TO_STRB(DALIShowShortAdr.wShortAddress_16_1));
		cmd := CONCAT(cmd, WORD_TO_STRB(DALIShowShortAdr.wShortAddress_32_17));
		cmd := CONCAT(cmd, WORD_TO_STRB(DALIShowShortAdr.wShortAddress_48_33));
		cmd := CONCAT(cmd, WORD_TO_STRB(DALIShowShortAdr.wShortAddress_64_49));
		start_send := TRUE;
		DaliSendAction := 0;
	ELSE
		DALIShowShortAdr(xQuery := TRUE);
	END_IF
*)
1: (* WAGO_DALI_GET_ADDR *)
	IF (dali_master = FALSE) THEN
		addr_1_16 := SHL(DaliMasterAdv.bByte_3, 8) + DaliMasterAdv.bByte_1;
		addr_17_32 := SHL(DaliMasterAdv.bByte_5, 8) + DaliMasterAdv.bByte_4;
		dali_master := TRUE;
		DALIMasterAdv(xStartDaliMaster := dali_master, iCommand := 507);
		DaliSendAction := 111;
	ELSE
		DaliMasterAdv(xStartDaliMaster := dali_master);
	END_IF
111: (* WAGO_DALI_GET_ADDR bis *)
	IF (dali_master = FALSE) THEN
		cmd := 'WAGO_DALI_GET_ADDR ';
		cmd := CONCAT(cmd, WORD_TO_STRB(addr_1_16));
		cmd := CONCAT(cmd, WORD_TO_STRB(addr_17_32));
		cmd := CONCAT(cmd, WORD_TO_STRB( SHL(DaliMasterAdv.bByte_3, 8) + DaliMasterAdv.bByte_1 ));
		cmd := CONCAT(cmd, WORD_TO_STRB( SHL(DaliMasterAdv.bByte_5, 8) + DaliMasterAdv.bByte_4 ));
		start_send := TRUE;
		DaliSendAction := 0;
	ELSE
		DaliMasterAdv(xStartDaliMaster := dali_master);
	END_IF
2: (* WAGO_DALI_GET_DEVICE_INFO *)
	IF (DALIConfigDevice.xReady = TRUE) THEN
		cmd := 'WAGO_DALI_GET_DEVICE_INFO ';
		cmd := CONCAT(cmd, WORD_TO_STRING(DALIConfigDevice.bFadeRate));
		cmd := CONCAT(cmd, ' ');
		cmd := CONCAT(cmd, WORD_TO_STRING(DALIConfigDevice.bFadeTime));
		cmd := CONCAT(cmd, ' ');
		cmd := CONCAT(cmd, WORD_TO_STRING(DALIConfigDevice.bMaxLevel));
		cmd := CONCAT(cmd, ' ');
		cmd := CONCAT(cmd, WORD_TO_STRING(DALIConfigDevice.bMinLevel));
		cmd := CONCAT(cmd, ' ');
		cmd := CONCAT(cmd, WORD_TO_STRING(DALIConfigDevice.bSystemFailureLevel));
		cmd := CONCAT(cmd, ' ');
		cmd := CONCAT(cmd, WORD_TO_STRING(DALIConfigDevice.bPowerOnLevel));
		start_send := TRUE;
		DaliSendAction := 0;
	ELSE
		DALIConfigDevice(xQuery := TRUE);
	END_IF
3: (* WAGO_DALI_GET_DEVICE_GROUP *)
	IF (dali_master = FALSE) THEN
		groups_cmd_1_8 := DaliMaster.bQueryValue;
		dali_master := TRUE;
		DALIMaster(xStartDaliMaster := dali_master, iCommand := 193, bAddress := group_address);
		DaliSendAction := 4;
	ELSE
		DaliMaster(xStartDaliMaster := dali_master);
	END_IF
4: (* WAGO_DALI_GET_DEVICE_GROUP bis *)
	IF (dali_master = FALSE) THEN
		cmd := 'WAGO_DALI_GET_DEVICE_GROUP ';
		cmd := CONCAT(cmd, BYTE_TO_STRING(group_address));
		cmd := CONCAT(cmd, ' ');
		cmd := CONCAT(cmd, WORD_TO_STRB( SHL(DaliMaster.bQueryValue, 8) + groups_cmd_1_8 ));
		start_send := TRUE;
		DaliSendAction := 0;
	ELSE
		DaliMaster(xStartDaliMaster := dali_master);
	END_IF
5: (* WAGO_DALI_DEVICE_ADD_GROUP *)
	IF (dali_master = FALSE) THEN
		cmd := 'WAGO_DALI_DEVICE_ADD_GROUP 1';
		start_send := TRUE;
		DaliSendAction := 0;
	ELSE
		DALIMasterAdv(xStartDaliMaster := dali_master);
	END_IF
6: (* WAGO_DALI_DEVICE_DEL_GROUP *)
	IF (dali_master = FALSE) THEN
		cmd := 'WAGO_DALI_DEVICE_DEL_GROUP 1';
		start_send := TRUE;
		DaliSendAction := 0;
	ELSE
		DALIMasterAdv(xStartDaliMaster := dali_master);
	END_IF
98: (* WAGO_DALI_ADDRESSING_STATUS *)
	IF (DALIConfigShortAddress.xReady = TRUE) THEN
		cmd := 'WAGO_DALI_ADDRESSING_STATUS 1';
		start_send := TRUE;
		DaliSendAction := 0;
	ELSE
		cmd := 'WAGO_DALI_ADDRESSING_STATUS 0';
		start_send := TRUE;
		DaliSendAction := 99;
		DALIConfigShortAddress(xNewAddressing := newAddressing, xExtendedAddressing := extendedAddr,
							   xReset := resetAddr, xSwitchAtAddressing := TRUE,
							   xReplaceShortAddress := replaceAddr, bOldShortAddress := oldAddr, bNewShortAddress := newAddr,
							   xDeleteShortAddress := delAddressing, bDeleteShortAddress := delAddr);
	END_IF
99: (* Addressing in progress *)
		DALIConfigShortAddress(xNewAddressing := newAddressing, xExtendedAddressing := extendedAddr,
							   xReset := resetAddr, xSwitchAtAddressing := TRUE,
							   xReplaceShortAddress := replaceAddr, bOldShortAddress := oldAddr, bNewShortAddress := newAddr,
							   xDeleteShortAddress := delAddressing, bDeleteShortAddress := delAddr);
END_CASE

IF (DaliSend = TRUE) THEN
	IF (dmx_read_addr > 0) THEN

		cmd := 'WAGO_DALI_GET ';
		IF (abDMX_Values[dmx_read_addr] < 1) THEN
			cmd := CONCAT(cmd, '0 ');
		ELSE
			cmd := CONCAT(cmd, '1 ');
		END_IF
		cmd := CONCAT(cmd, ITOA(BYTE_TO_INT(abDMX_Values[dmx_read_addr] * 100 / 255)));
		start_send := TRUE;
		DaliSend := FALSE;
	ELSE
		IF (DALIDimmValue.xReady = TRUE) THEN
			cmd := 'WAGO_DALI_GET ';
			cmd := CONCAT(cmd, ITOA(BOOL_TO_INT(DALIDimmValue.xStatus)));
			cmd := CONCAT(cmd, ' ');
			cmd := CONCAT(cmd, ITOA(BYTE_TO_INT(DALIDimmValue.bDimmValue)));
			start_send := TRUE;
			DaliSend := FALSE;
		ELSE
			DALIDimmValue(xEnable := TRUE, bShortAddress := DINT_TO_BYTE(p2), tCycleTime := t#1s);
		END_IF
	END_IF
END_IF

IF (HEARTBEAT_TIMER.Q = TRUE) THEN
	(* We lost the connection with the server *)
	(* The wago is now in standalone mode *)
	HEARTBEAT := FALSE;

	LedMode := 1;
ELSE
	HEARTBEAT := TRUE;
END_IF
END_PROGRAM

(* POU EthernetServer_FB, ST *)
FUNCTION_BLOCK EthernetServer_FB
(************************************************************)
(* ETHERNET_SERVER		                          		    *)
(* Ver. 1.0   	                                         	*)
(* Date:  10.02.2003					         	 		*)
(* Author:  Volker Begemann                            		*)
(************************************************************)
VAR_INPUT
	xOPEN_SERVER		:	BOOL;				(* Set TRUE to enable function block			*)
	wPORT					:	WORD;				(* Port number											*)
	xTCP_PROTOCOL		:	BOOL;				(* TRUE => TCP; FALSE => UDP						*)
	tTIMEOUT				:	TIME:=t#20s;	(* Watchdog timeout value (seconds)				*)
	iBYTES_TO_SEND		:	INT;				(* Number of bytes to transmit					*)
	ptSEND_BUFFER		:	POINTER TO ARRAY[1..1500] OF BYTE;		(* Transmit Buffer	*)
END_VAR
VAR_IN_OUT
	xSTART_SEND:		BOOL;						(* Set TRUE to initiate data transmittal, will be	*)
														(* reset FALSE when transmittal is completed 		*)
(* 	utRECEIVE_BUFFER:	typEthernetBuffer;	(* Receive Buffer *) *)
	ptRECV_BUFFER		:	POINTER TO ARRAY[1..1500] OF BYTE;		(* Receive Buffer	*)
END_VAR
VAR_OUTPUT
	utERROR					:	ETH_ERROR;	(* See ETH_ERROR datatype in ETHERNET.LIB	*)
													(* for error codes and definitions			*)
	xSERVER_OPEN:			BOOL;				(* TRUE if socket connection made			*)
	wSOCKET:					WORD;				(* Socket connection number					*)
	bDataReceived: 		BOOL := FALSE;
	iBYTES_RECEIVED: INT; (* Number of bytes received *)
END_VAR
VAR
	i: INT;
	CloseState:			INT;
	EthernetOpen:		ETHERNET_SERVER_OPEN;
	EthernetClose:		ETHERNET_SERVER_CLOSE;
	EthernetWrite:		ETHERNET_WRITE;
	EthernetRead:		ETHERNET_READ;
	GetConfig:			ETHERNET_GET_NETWORK_CONFIG;
	EthernetBuffer:	ARRAY[1..1500] OF BYTE;
	Status:				WORD:=0;
	client_SRC_PORT:	WORD;
	watchdog_timer1:	TON;
	client_SRC_IP:		DWORD;
END_VAR
IF xOPEN_SERVER THEN
	watchdog_timer1(IN:=TRUE , PT:=tTIMEOUT );

	IF watchdog_timer1.q THEN
		watchdog_timer1(IN:=FALSE , PT:=tTIMEOUT );
		EthernetClose(EN:= 1, SOCKET:= EthernetOpen.SOCKET);
		EthernetClose(EN:= 0, SOCKET:= 0);
		Status := 0; (* Try to open the server *)
	END_IF

	CASE Status OF
		0:
			GetConfig(EN:=FALSE );
			GetConfig(EN:=TRUE );
			utERROR		:=	0;
			wSocket		:=	0;
			CloseState	:=	0;
			status		:=	1;
		1:
			GetConfig(EN:=TRUE );
			IF GetConfig.ENO THEN
				IF GetConfig.IP_ADR<>0 THEN
					status:=4;
					EthernetOpen (EN:=0);
					EthernetRead(EN:= 0, SOCKET:=0 ,  DATA:=EthernetBuffer );
					EthernetClose(EN:= 0);
				ELSE
					status:=0;
				END_IF
			END_IF
		4: 	(* try to open a socket*)
			IF xTCP_PROTOCOL THEN
				EthernetOpen(EN:=1 , TYP:=SOCK_STREAM, PROTO := IPPROTO_TCP, PORT := wPort);
			ELSE
				EthernetOpen(EN:=1 , TYP:=SOCK_DGRAM, PROTO := IPPROTO_UDP, PORT := wPort);
			END_IF
			IF ((EthernetOpen.ERROR = 0) AND (EthernetOpen.ENO = 1)) THEN
				Status  := 10; (* socket created, wait for data to process *)
				EthernetOpen (EN:=0);
				xServer_open:=TRUE;
				wSocket:=EthernetOpen.socket;
			ELSE
				Status := 0; 	(* socket not available, try it again *)
				EthernetOpen (EN:=0);
				xServer_open:=FALSE;
				wSocket:=0;
			END_IF;

		10: 	(* Wait for data to process *)
			(* Monitor ethernet port for new data *)
			bDataReceived	:= FALSE;
	 		EthernetRead(	EN:= 1, SOCKET:=EthernetOpen.SOCKET, DATA:=EthernetBuffer);
			EthernetRead(	EN:= 0, SOCKET:=0, DATA:=EthernetBuffer);

			IF(EthernetRead.ERROR<>0) THEN  			(* Error reading the socket, close it *)
				Status	:=	40;
			ELSIF (EthernetRead.LEN_OUT <>0) THEN  (* Process the data received via the ethernet port *)
				client_SRC_IP		:=	EthernetRead.SRC_IP;
				client_SRC_PORT	:=	EthernetRead.SRC_PORT;
				ptRECV_BUFFER^		:= EthernetBuffer;
				bDataReceived		:= TRUE;
				iBYTES_RECEIVED		:= EthernetRead.LEN_OUT;
				watchdog_timer1(IN:=FALSE, PT:=tTIMEOUT );
			ELSIF (iBytes_TO_SEND > 0 AND xSTART_SEND) THEN  (* Process the data received *)
				EthernetWrite(EN:= 0, DATA:=EthernetBuffer);
				status	:=	30;
			END_IF

		30: 	(* Process the data to send *)
			EthernetBuffer :=ptSEND_BUFFER^;
			(* Send data in transmit buffer out ethernet port *)
			IF xTCP_PROTOCOL THEN
					EthernetWrite(	EN:= 1,
								SOCKET:= EthernetOpen.SOCKET,
								LEN_IN:=iBYTES_TO_SEND,
								DATA:=EthernetBuffer );
			ELSE
				IF client_SRC_IP>0 AND client_SRC_PORT>0 THEN
					EthernetWrite(EN:=1, SOCKET:=EthernetOpen.SOCKET , LEN_IN:=iBYTES_TO_SENd , DST_IP:=client_SRC_IP,DST_PORT:=client_SRC_PORT,DATA:=EthernetBuffer );
				ELSE
					status:=10;
				END_IF
			END_IF

			IF EthernetWrite.eno THEN
				IF(EthernetWrite.ERROR <>0) THEN
					Status:=40;(* Error writing to the socket, close it *)
				ELSE
					Status:=10; (* Comms complete, read more data *)
				END_IF;
				xStart_send:=FALSE;
			END_IF
		40:	(* Close the server *)
			EthernetClose(EN:= 1, SOCKET:= EthernetOpen.SOCKET);
			IF EthernetClose.eno THEN
				EthernetClose(EN:= 0);
				xOPEN_SERVER:=FALSE;
				utERROR:=0;
				wSocket:=0;
				Status := 0; (* Try to open the server again *)
			END_IF

	END_CASE;
ELSE
	CASE CloseState OF
	0:
		EthernetClose(EN:= 0);
		EthernetClose(EN:= 1, SOCKET:= EthernetOpen.SOCKET);
		CloseState:=1;
	1:
		EthernetClose(EN:= 1, SOCKET:= EthernetOpen.SOCKET);
		IF EthernetClose.eno THEN
			EthernetClose(EN:= 0);
			CloseState:=2;
		END_IF
	2:
		xOPEN_SERVER:=FALSE;
		utERROR:=0;
		wSocket:=0;
	END_CASE
END_IF
END_FUNCTION_BLOCK

(* POU Strncmp, ST *)
FUNCTION Strncmp : BOOL
VAR_INPUT
	str1: STRING;
	str2: STRING;
	n: BYTE;
END_VAR
VAR
	tmp1: POINTER TO ARRAY[0..255] OF BYTE;
	tmp2: POINTER TO ARRAY[0..255] OF BYTE;
	i: BYTE;
END_VAR
tmp1 := ADR(str1);
tmp2 := ADR(str2);

Strncmp := TRUE;

FOR i := 0 TO n - 1 DO
	IF (tmp1^[i] <> tmp2^[i]) THEN
		Strncmp := FALSE;
		i := n;
	END_IF
END_FOR
END_FUNCTION

(* POU GET_PARAM_DINT, ST *)
FUNCTION GET_PARAM_DINT : DINT
VAR_INPUT
	str: STRING;
	pos: BYTE;
END_VAR
VAR
	i: BYTE;
	j: BYTE;
	mult : DWORD;
	dec : DWORD;
	p: INT;
	tmp: POINTER TO ARRAY[0..255] OF BYTE;
	val: DINT;
	neg: BOOL := FALSE;
END_VAR
(* cut before the value we want *)
FOR i := 1 TO pos DO
	str := DELETE(str, FIND(str, ' '), 1);
END_FOR

(* cut after the value we want *)
p := FIND(str, ' ');
IF (p > 0) THEN
	str := LEFT(str, p - 1);
END_IF

(* Convert the value *)
tmp := ADR(str);

IF (Strncmp(str, '-', 1) = TRUE) THEN
	neg := TRUE;
	str := DELETE(str, 1, 1);
END_IF

val := 0;
FOR i := 0 TO INT_TO_BYTE(LEN(str) - 1) DO
	dec := 1;
	FOR j := 2 TO INT_TO_BYTE(LEN(str) - i) DO
		dec := dec * 10;
	END_FOR

	mult := tmp^[i] - 16#30;
	mult := mult * dec;
	val := val + mult;

END_FOR

IF (neg = TRUE) THEN
	GET_PARAM_DINT := 0 - val;
ELSE
	GET_PARAM_DINT := val;
END_IF
END_FUNCTION

(* POU VOLET, ST *)
FUNCTION_BLOCK VOLET
VAR
	sens: BOOL;
	imp: TP;
	mode: VOLET_MODE;
END_VAR
VAR_INPUT
	IN: BOOL;
	IMPULSE: BOOL;
END_VAR
VAR_OUTPUT
	MONTE: BOOL;
	DESCENTE:BOOL;
END_VAR
(* Volet *)

IF IMPULSE = FALSE THEN
	(* Normal mode *)
	IF (MONTE = TRUE OR DESCENTE = TRUE) THEN
		MONTE := FALSE;
		DESCENTE := FALSE;
	ELSE

		IF IN = TRUE THEN
			IF sens = TRUE THEN
				sens := FALSE;
			ELSE
				sens := TRUE;
			END_IF;

			IF sens = TRUE THEN
				(*monte*)
				DESCENTE := FALSE;
				MONTE := TRUE;
			ELSE
				MONTE := FALSE;
				DESCENTE := TRUE;
			END_IF;
		END_IF

	END_IF
ELSE
	(* impulse mode *)
	imp(IN := FALSE, PT:= impulse_time);

	IF mode = IMP_STOP THEN
		MONTE := imp.Q;
		DESCENTE := imp.Q;
		IF imp.Q = FALSE THEN
			mode := VOLET_STOP;
		END_IF;
	END_IF;
	IF mode = IMP_UP THEN
		MONTE := imp.Q;
		DESCENTE := FALSE;
		IF imp.Q = FALSE THEN
			mode := VOLET_UP;
		END_IF;
	END_IF;
	IF mode = IMP_DOWN THEN
		MONTE := FALSE;
		DESCENTE := imp.Q;
		IF imp.Q = FALSE THEN
			mode := VOLET_DOWN;
		END_IF;
	END_IF;

	IF mode = VOLET_UP OR mode = VOLET_DOWN THEN
		IF IN = TRUE THEN
			imp(IN := TRUE, PT:= impulse_time);
			mode := IMP_STOP;
		END_IF;
	ELSE
		IF IN = TRUE THEN
			IF sens = TRUE THEN
				sens := FALSE;
			ELSE
				sens := TRUE;
			END_IF;

			IF sens = TRUE THEN
				imp(IN := TRUE, PT:= impulse_time);
				mode := IMP_UP;
			ELSE
				imp(IN := TRUE, PT:= impulse_time);
				mode := IMP_DOWN;
			END_IF;
		END_IF;
	END_IF;
END_IF;
END_FUNCTION_BLOCK

(* POU ITOA, ST *)
FUNCTION ITOA : STRING
VAR_INPUT
	VAL: INT;
END_VAR
VAR
	tmp: INT;
	conv: INT;
END_VAR
(* Convert a byte to string *)

IF (VAL < 0) THEN
	tmp := -VAL;
ELSE
	tmp := VAL;
END_IF

IF (tmp = 0) THEN
	ITOA := ASCIIBYTE_TO_STRING(0 + 16#30);
END_IF

WHILE (tmp > 0) DO
	conv := tmp MOD 10;
	tmp := tmp / 10;
	ITOA := INSERT(ITOA, ASCIIBYTE_TO_STRING(INT_TO_BYTE(conv) + 16#30), 0);
END_WHILE

IF (VAL < 0) THEN
	ITOA := INSERT(ITOA, '-', 0);
END_IF
END_FUNCTION

(* POU DMX, FBD *)
PROGRAM DMX
VAR
	DMX_Master				: FbDMX_StageProfi;
		Enable				: BOOL := TRUE ;
		PortNumber			: WORD := 10001;
		FirstChannel		: WORD := 1;
		NumberOfChannels	: BYTE := 255;
		Ready				: BOOL;
		Connect				: BOOL;
		ErrorCode			: DINT;
		ErrorWatchdog		: BOOL;
END_VAR
VAR_INPUT RETAIN
		IPaddress			: STRING(16) := '192.168.1.120';
END_VAR
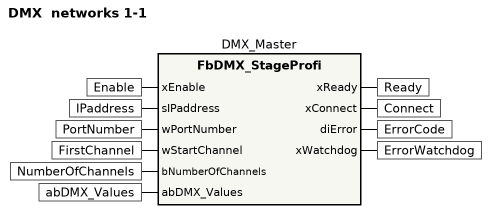
_FBD_ (* Function Block Diagram *)
NETWORK 1
	DMX_Master:FbDMX_StageProfi(xEnable: Enable, sIPaddress: IPaddress, wPortNumber: PortNumber, wStartChannel: FirstChannel, bNumberOfChannels: NumberOfChannels, abDMX_Values: abDMX_Values, xConnect => Connect, diError => ErrorCode, xWatchdog => ErrorWatchdog) => Ready
_END_FBD_
(* the same logic as Structured Text *)
(* Network 1 *)
DMX_Master(xEnable := Enable, sIPaddress := IPaddress, wPortNumber := PortNumber, wStartChannel := FirstChannel, bNumberOfChannels := NumberOfChannels, abDMX_Values := abDMX_Values);
Connect := DMX_Master.xConnect;
ErrorCode := DMX_Master.diError;
ErrorWatchdog := DMX_Master.xWatchdog;
Ready := DMX_Master.xReady;
END_PROGRAM

(* POU SetOutput, ST *)
FUNCTION SetOutput : BOOL
VAR_INPUT
	bit_offset: UINT;
	val: BOOL;
END_VAR
VAR
END_VAR
(* Set the bit in OutArrState Array *)

IF (val = TRUE) THEN
	OutArrState[bit_offset / 8] := OutArrState[bit_offset / 8] OR SHL(16#01, bit_offset MOD 8);
ELSE
	OutArrState[bit_offset / 8] := OutArrState[bit_offset / 8] AND NOT SHL(16#01, bit_offset MOD 8);
END_IF

SetOutput := TRUE;
END_FUNCTION

(* POU WORD_TO_STRB, ST *)
FUNCTION WORD_TO_STRB : STRING(16)
VAR_INPUT
	IN : WORD;
END_VAR
VAR
	pt : POINTER TO BYTE;
	i: INT;
END_VAR
pt := ADR(WORD_TO_STRB);

FOR i := 1 TO 16 DO
	pt^:= BOOL_TO_BYTE(in.0) + 48;
	in := SHR(in,1);
	pt := pt + 1;
END_FOR;

pt^ := 0;
END_FUNCTION

(* POU ManageOutput, ST *)
PROGRAM ManageOutput
VAR
	cpt: INT;
	tmp: INT;
	_light: LIGHT;
	in: BOOL;
END_VAR
(* Set all outputs when in standalone mode *)

(* Get the address of the first digital output *)
FOR cpt := 0 TO 512 DO

	CASE output_type[cpt] OF
	NONE: (* Do nothing *);
	TELERUPTEUR:
		tmp := cpt;
		IF (output_addr[cpt].SameAs >= 0) THEN
			tmp := output_addr[cpt].SameAs;
		END_IF
		IF (event[cpt].ON = TRUE) THEN
			_light(IN := FALSE, STATE := BYTE_TO_BOOL(SHR(lights[tmp / 8], tmp MOD 8) AND 16#01));
			_light(IN := TRUE, STATE := BYTE_TO_BOOL(SHR(lights[tmp / 8], tmp MOD 8) AND 16#01));
			SetOutput(output_addr[tmp].ADDR1 + start_addr_out, _light.OUT);

			(* set old state *)
			IF (_light.OUT = TRUE) THEN
				lights[tmp / 8] := lights[tmp / 8] OR SHL(16#01, tmp MOD 8);
			ELSE
				lights[tmp / 8] := lights[tmp / 8] AND NOT SHL(16#01, tmp MOD 8);
			END_IF
		END_IF
	DIRECT:
		tmp := cpt;
		IF (output_addr[cpt].SameAs >= 0) THEN
			tmp := output_addr[cpt].SameAs;
		END_IF
		IF (cpt >= 256) THEN
			; (* knx only *)
		ELSE
			in := GetInput(cpt + start_addr_in);
		END_IF
		SetOutput(output_addr[tmp].ADDR1 + start_addr_out, in);
	VOLET:
		tmp := cpt;
		IF (output_addr[cpt].SameAs >= 0) THEN
			tmp := output_addr[cpt].SameAs;
		END_IF
		IF (event[cpt].ON = TRUE) THEN
			volets[tmp](IN := TRUE, IMPULSE := FALSE);
			SetOutput(output_addr[tmp].ADDR1 + start_addr_out, volets[tmp].MONTE);
			SetOutput(output_addr[tmp].ADDR2 + start_addr_out, volets[tmp].DESCENTE);
		END_IF
	VOLET_IMPULSE:
		tmp := cpt;
		IF (output_addr[cpt].SameAs >= 0) THEN
			tmp := output_addr[cpt].SameAs;
		END_IF
		IF (event[cpt].ON = TRUE) THEN
			volets[tmp](IN := TRUE, IMPULSE := TRUE);
		ELSE
			volets[tmp](IN := FALSE, IMPULSE := TRUE);
		END_IF
		SetOutput(output_addr[tmp].ADDR1 + start_addr_out, volets[tmp].MONTE);
		SetOutput(output_addr[tmp].ADDR2 + start_addr_out, volets[tmp].DESCENTE);
	TELERUPTEUR_DALI:
		tmp := cpt;
		IF (output_addr[cpt].SameAs >= 0) THEN
			tmp := output_addr[cpt].SameAs;
		END_IF
		IF (event[cpt].ON = TRUE) THEN
			_light(IN := FALSE, STATE := BYTE_TO_BOOL(SHR(lights[tmp / 8], tmp MOD 8) AND 16#01));
			_light(IN := TRUE, STATE := BYTE_TO_BOOL(SHR(lights[tmp / 8], tmp MOD 8) AND 16#01));

			IF (output_addr[tmp].ADDR2 > 99) THEN
				IF (_light.OUT = TRUE) THEN
					abDMX_Values[WORD_TO_BYTE(output_addr[tmp].ADDR2 - 100)] := 255;
				ELSE
					abDMX_Values[WORD_TO_BYTE(output_addr[tmp].ADDR2 - 100)] := 0;
				END_IF
			ELSE
				Dali_switch(xButton := FALSE);
				IF (_light.OUT = TRUE) THEN
					Dali_switch(bAddress := WORD_TO_BYTE(output_addr[tmp].ADDR2), xGroup := FALSE, bDimmLevel := 100,
						bFadeTime := 1, xButton := TRUE);
				ELSE
					Dali_switch(bAddress := WORD_TO_BYTE(output_addr[tmp].ADDR2), xGroup := FALSE, bDimmLevel := 0,
						bFadeTime := 1, xButton := TRUE);
				END_IF
			END_IF

			(* set old state *)
			IF (_light.OUT = TRUE) THEN
				lights[tmp / 8] := lights[tmp / 8] OR SHL(16#01, tmp MOD 8);
			ELSE
				lights[tmp / 8] := lights[tmp / 8] AND NOT SHL(16#01, tmp MOD 8);
			END_IF
		END_IF
	TELERUPTEUR_DALI_GROUP:
		tmp := cpt;
		IF (output_addr[cpt].SameAs >= 0) THEN
			tmp := output_addr[cpt].SameAs;
		END_IF
		IF (event[cpt].ON = TRUE) THEN
			_light(IN := FALSE, STATE := BYTE_TO_BOOL(SHR(lights[tmp / 8], tmp MOD 8) AND 16#01));
			_light(IN := TRUE, STATE := BYTE_TO_BOOL(SHR(lights[tmp / 8], tmp MOD 8) AND 16#01));
			Dali_switch(xButton := FALSE);
			IF (_light.OUT = TRUE) THEN
				Dali_switch(bAddress := WORD_TO_BYTE(output_addr[tmp].ADDR2), xGroup := TRUE, bDimmLevel := 100,
					bFadeTime := 1, xButton := TRUE);
			ELSE
				Dali_switch(bAddress := WORD_TO_BYTE(output_addr[tmp].ADDR2), xGroup := TRUE, bDimmLevel := 0,
					bFadeTime := 1, xButton := TRUE);
			END_IF

			(* set old state *)
			IF (_light.OUT = TRUE) THEN
				lights[tmp / 8] := lights[tmp / 8] OR SHL(16#01, tmp MOD 8);
			ELSE
				lights[tmp / 8] := lights[tmp / 8] AND NOT SHL(16#01, tmp MOD 8);
			END_IF
		END_IF
	TELERUPTEUR_KNX_OUTPUT:
		;(* Works only on 750-849 *)
	DIRECT_KNX_OUTPUT:
		;(* Works only on 750-849 *)

	END_CASE
END_FOR
END_PROGRAM

(* POU LIGHT, ST *)
FUNCTION_BLOCK LIGHT
VAR
	TRIG: R_TRIG;
	light: BOOL;
END_VAR
VAR_INPUT
	IN: BOOL;
	STATE: BOOL;
END_VAR
VAR_OUTPUT
	OUT: BOOL;
END_VAR
(* telerupteur *)

TRIG(CLK := IN);
light := TRIG.Q;

OUT := STATE;

IF light = TRUE THEN
	IF OUT = TRUE THEN
		OUT := FALSE;
	ELSE
		OUT := TRUE;
	END_IF;
END_IF;
END_FUNCTION_BLOCK

(* POU DMX_Fading_Task, ST *)
PROGRAM DMX_Fading_Task
VAR
	fade: DMX_Fade;
	t: BOOL := FALSE;
END_VAR
(*
IF (NOT t) THEN
		abDMX_Values[1] := 200;
		fade(xEnable := FALSE);
		fade(xEnable := TRUE, DMXAddr := 1, DMXNewValue := 40);
		t := TRUE;
END_IF

fade();
*)
;
END_PROGRAM

(* POU DMX_Fade, ST *)
FUNCTION_BLOCK DMX_Fade
VAR_INPUT
	xEnable: BOOL;
	DMXAddr: BYTE;
	DMXNewValue: BYTE;
END_VAR
VAR_OUTPUT
	xReady: BOOL := TRUE;
END_VAR
VAR
	Mtrig: R_TRIG;
	value: INT;
	act: BYTE;
	dtime: INT;
	DMXold: INT;
	currentTimeFB: CurTime;
	currentTime, startTime: SysTime64;
END_VAR
VAR CONSTANT
	FadeTime: WORD := 500; (* Fade time in ms *)
	FadeStep: WORD := 30;  (* Fade step in ms *)
END_VAR
Mtrig(CLK := xEnable);
IF (Mtrig.Q = TRUE) THEN
	xReady := FALSE;
	dtime := 0;
	DMXold := abDMX_Values[DMXAddr];

	IF (DMXold < DMXNewValue) THEN
		act := 1;
	ELSE
		act := 2;
	END_IF

	currentTimeFB(SystemTime := startTime);

END_IF

IF (xReady = TRUE) THEN
	RETURN;
END_IF

IF (dtime >= FadeTime) THEN
	xReady := TRUE;
	RETURN;
END_IF

dtime := dtime + FadeStep;

IF (dtime > FadeTime) THEN
	dtime := FadeTime;
END_IF

CASE act OF

1: (* up *)
	value := DMXold + dtime * (BYTE_TO_INT(DMXNewValue) - DMXold) / FadeTime;
	IF (value > DMXNewValue) THEN
		value := DMXNewValue;
		xReady := TRUE;
	END_IF

	abDMX_Values[DMXAddr] := INT_TO_BYTE(value);

2: (* down *)
	value := DMXold + dtime * (BYTE_TO_INT(DMXNewValue) - DMXold) / FadeTime;
	IF (value < DMXNewValue) THEN
		value := DMXNewValue;
		xReady := TRUE;
	END_IF

	abDMX_Values[DMXAddr] := INT_TO_BYTE(value);

END_CASE
END_FUNCTION_BLOCK

(* POU INTER_EVENT, ST *)
FUNCTION_BLOCK INTER_EVENT
VAR_INPUT
	IN: BOOL;
END_VAR
VAR_OUTPUT
	ON: BOOL;
	OFF: BOOL;
END_VAR
VAR
	MTRIG: R_TRIG;
	DTRIG: F_TRIG;
END_VAR
(* Get the ON or OFF event on an input *)

MTRIG(CLK := IN);
ON := MTRIG.Q;
DTRIG(CLK := IN);
OFF := DTRIG.Q;
END_FUNCTION_BLOCK

(* Visualisation Addressing
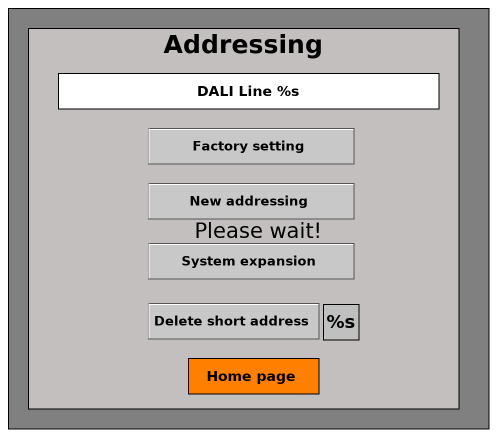
rectangle at (185,80)-(616,461): text "Addressing"
button at (305,235)-(511,271): text "New addressing"; taps DALI_Config.NewAddress; tooltip You have to click and hold the button "New Addressing" longer than two seconds to start the new addressing.
button at (305,295)-(511,331): text "System expansion"; taps DALI_Config.xErweitert; tooltip If you click the button "System expansion", only the ECGs with no short address will be addressed.
rectangle at (480,356)-(516,392): text "%s"; shows DALI_Config.LoeschKurzadr; tooltip Enter the short address to be deleted (1 - 64).; editable
rounded rectangle at (345,410)-(476,446): text "Home page"; opens PLC_VISU; tooltip Back to home page
button at (305,180)-(511,216): text "Factory setting"; taps DALI_Config.Reset; tooltip To reset the ECG you have to click and hold the button two seconds. Group and scene configurations will be deleted.
button at (305,355)-(476,391): text "Delete short address"; taps DALI_Config.Loeschen; tooltip The selected short address will be deleted.
rectangle at (275,97)-(556,468): text "Please wait!"; invisible if not DALI_Config.JobMerker[5]
rounded rectangle at (215,125)-(596,161): text "DALI Line %s"; shows DALI_Config.bDali_Linie; tooltip You can change the DALI Line only on the home page.
1 more shapes without text or variables
*)

(* Visualisation ECG_settings
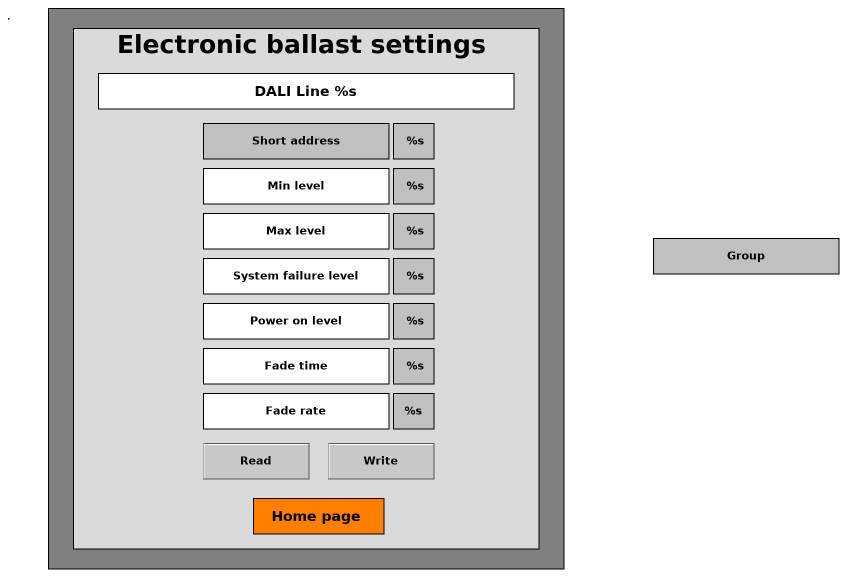
rectangle at (150,40)-(616,561): text "Electronic ballast settings"
rectangle at (280,225)-(466,261): text "Max level"
rectangle at (280,180)-(466,216): text "Min level"
rectangle at (280,270)-(466,306): text "System failure level"
rectangle at (280,315)-(466,351): text "Power on level"
rectangle at (280,360)-(466,396): text "Fade time"
rectangle at (280,405)-(466,441): text "Fade rate"
rectangle at (280,135)-(466,171): text "Short address"; invisible if DALI_Config.Kurzadr_Gruppe; toggles DALI_Config.Kurzadr_Gruppe
rectangle at (730,250)-(916,286): text "Group"; invisible if not DALI_Config.Kurzadr_Gruppe; toggles DALI_Config.Kurzadr_Gruppe; tooltip Selection group or short address
rectangle at (470,135)-(511,171): text "%s"; shows DALI_Config.Adresse; tooltip Enter group (1-16) or short address (1 - 64); editable
rounded rectangle at (330,510)-(461,546): text "Home page"; opens PLC_VISU; tooltip Back to home page
rectangle at (470,180)-(511,216): text "%s"; shows DALI_Config.MinLevel; tooltip Minimal brightness level in percent. Min level has to be smaller than max level.; editable
rectangle at (470,225)-(511,261): text "%s"; shows DALI_Config.MaxLevel; tooltip Maximum brightness level in percent; editable
rectangle at (470,270)-(511,306): text "%s"; shows DALI_Config.SystemFailure; tooltip Brightness level in percent in case of a system failure. The value 101 means "MASK".; editable
rectangle at (470,315)-(511,351): text "%s"; shows DALI_Config.PowerOn; tooltip Brightness level in percent if the ECGs are powered on.; editable
rectangle at (470,360)-(511,396): text "%s"; shows DALI_Config.Konfig[4]; tooltip Enter the fade time (0 - 15); editable
rectangle at (470,405)-(511,441): text "%s"; shows DALI_Config.Konfig[5]; tooltip Enter the fade rate (1 -15); editable
button at (280,455)-(386,491): text "Read"; taps DALI_Config.Lese; tooltip If you click the button "Read", the settings of the ECG will be read. Group queries are not possible.
button at (405,455)-(511,491): text "Write"; taps DALI_Config.Schreib; tooltip If you click the button "Write", the new settings will be written into the ECG.
rounded rectangle at (175,85)-(591,121): text "DALI Line %s"; shows DALI_Config.bDali_Linie; tooltip You can change the DALI Line only on the home page.
2 more shapes without text or variables
*)

(* Visualisation Group_assignment
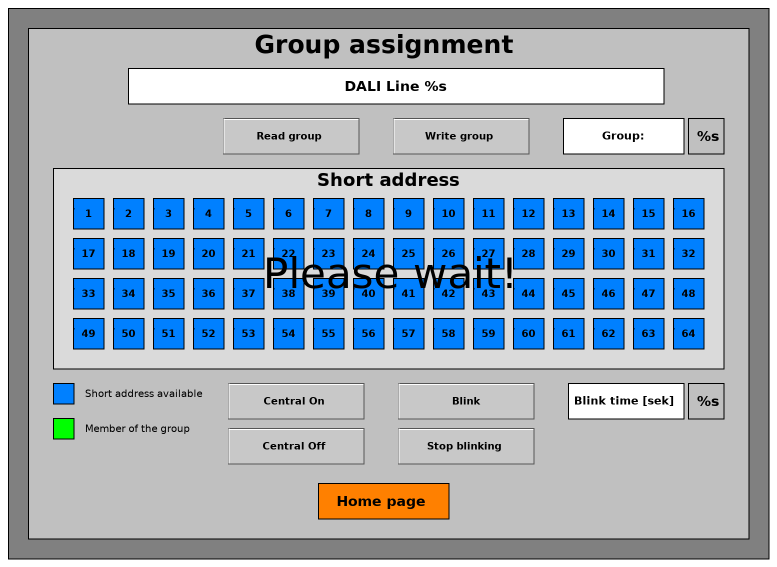
rectangle at (40,40)-(761,551): text "Group assignment"
rounded rectangle at (330,495)-(461,531): text "Home page"; opens PLC_VISU; tooltip Back to home page
rectangle at (65,180)-(736,381): text "Short address"
rectangle at (85,210)-(116,241): text "1"; alarm colour if DALI_Config.Kurzadr[1]
rectangle at (85,210)-(116,241): text "1"; invisible if not DALI_Config.Kurzadr[1]; alarm colour if DALI_Config.Gruppenadr[1]; toggles DALI_Config.Gruppenadr[1]
rectangle at (125,210)-(156,241): text "2"; alarm colour if DALI_Config.Kurzadr[2]
rectangle at (125,210)-(156,241): text "2"; invisible if not DALI_Config.Kurzadr[2]; alarm colour if DALI_Config.Gruppenadr[2]; toggles DALI_Config.Gruppenadr[2]
rectangle at (165,210)-(196,241): text "3"; alarm colour if DALI_Config.Kurzadr[3]
rectangle at (165,210)-(196,241): text "3"; invisible if not DALI_Config.Kurzadr[3]; alarm colour if DALI_Config.Gruppenadr[3]; toggles DALI_Config.Gruppenadr[3]
rectangle at (205,210)-(236,241): text "4"; alarm colour if DALI_Config.Kurzadr[4]
rectangle at (205,210)-(236,241): text "4"; invisible if not DALI_Config.Kurzadr[4]; alarm colour if DALI_Config.Gruppenadr[4]; toggles DALI_Config.Gruppenadr[4]
rectangle at (245,210)-(276,241): text "5"; alarm colour if DALI_Config.Kurzadr[5]
rectangle at (245,210)-(276,241): text "5"; invisible if not DALI_Config.Kurzadr[5]; alarm colour if DALI_Config.Gruppenadr[5]; toggles DALI_Config.Gruppenadr[5]
rectangle at (285,210)-(316,241): text "6"; alarm colour if DALI_Config.Kurzadr[6]
rectangle at (285,210)-(316,241): text "6"; invisible if not DALI_Config.Kurzadr[6]; alarm colour if DALI_Config.Gruppenadr[6]; toggles DALI_Config.Gruppenadr[6]
rectangle at (325,210)-(356,241): text "7"; alarm colour if DALI_Config.Kurzadr[7]
rectangle at (325,210)-(356,241): text "7"; invisible if not DALI_Config.Kurzadr[7]; alarm colour if DALI_Config.Gruppenadr[7]; toggles DALI_Config.Gruppenadr[7]
rectangle at (365,210)-(396,241): text "8"; alarm colour if DALI_Config.Kurzadr[8]
rectangle at (365,210)-(396,241): text "8"; invisible if not DALI_Config.Kurzadr[8]; alarm colour if DALI_Config.Gruppenadr[8]; toggles DALI_Config.Gruppenadr[8]
rectangle at (405,210)-(436,241): text "9"; alarm colour if DALI_Config.Kurzadr[9]
rectangle at (405,210)-(436,241): text "9"; invisible if not DALI_Config.Kurzadr[9]; alarm colour if DALI_Config.Gruppenadr[9]; toggles DALI_Config.Gruppenadr[9]
rectangle at (445,210)-(476,241): text "10"; alarm colour if DALI_Config.Kurzadr[10]
rectangle at (445,210)-(476,241): text "10"; invisible if not DALI_Config.Kurzadr[10]; alarm colour if DALI_Config.Gruppenadr[10]; toggles DALI_Config.Gruppenadr[10]
rectangle at (485,210)-(516,241): text "11"; alarm colour if DALI_Config.Kurzadr[11]
rectangle at (485,210)-(516,241): text "11"; invisible if not DALI_Config.Kurzadr[11]; alarm colour if DALI_Config.Gruppenadr[11]; toggles DALI_Config.Gruppenadr[11]
rectangle at (525,210)-(556,241): text "12"; alarm colour if DALI_Config.Kurzadr[12]
rectangle at (525,210)-(556,241): text "12"; invisible if not DALI_Config.Kurzadr[12]; alarm colour if DALI_Config.Gruppenadr[12]; toggles DALI_Config.Gruppenadr[12]
rectangle at (565,210)-(596,241): text "13"; alarm colour if DALI_Config.Kurzadr[13]
rectangle at (565,210)-(596,241): text "13"; invisible if not DALI_Config.Kurzadr[13]; alarm colour if DALI_Config.Gruppenadr[13]; toggles DALI_Config.Gruppenadr[13]
rectangle at (605,210)-(636,241): text "14"; alarm colour if DALI_Config.Kurzadr[14]
rectangle at (605,210)-(636,241): text "14"; invisible if not DALI_Config.Kurzadr[14]; alarm colour if DALI_Config.Gruppenadr[14]; toggles DALI_Config.Gruppenadr[14]
rectangle at (645,210)-(676,241): text "15"; alarm colour if DALI_Config.Kurzadr[15]
rectangle at (645,210)-(676,241): text "15"; invisible if not DALI_Config.Kurzadr[15]; alarm colour if DALI_Config.Gruppenadr[15]; toggles DALI_Config.Gruppenadr[15]
rectangle at (685,210)-(716,241): text "16"; alarm colour if DALI_Config.Kurzadr[16]
rectangle at (685,210)-(716,241): text "16"; invisible if not DALI_Config.Kurzadr[16]; alarm colour if DALI_Config.Gruppenadr[16]; toggles DALI_Config.Gruppenadr[16]
button at (405,130)-(541,166): text "Write group"; taps DALI_Config.Gruppenkonfiguration; tooltip If you click the button "Write Group", the marked short addresses will be saved as a group.
rectangle at (575,130)-(696,166): text "Group:"
rectangle at (700,130)-(736,166): text "%s"; shows DALI_Config.Gruppe; tooltip Enter the number of the group (1 - 16); editable
button at (410,395)-(546,431): text "Blink"; taps DALI_Config.BlinkenGruppe; tooltip If you click the button "Blink", the selected ECG will blink as long as defined by the "Blink Time" parameter.
button at (410,440)-(546,476): text "Stop blinking"; taps DALI_Config.xBlinken_Aus; tooltip If you click the button "Stop blinking", the blinking of the ECG will stop immediately.
button at (235,130)-(371,166): text "Read group"; taps DALI_Config.GruppeLesen; tooltip If you click the button "Read Group", the short addresses that belong to the group will be displayed.
rectangle at (95,395)-(226,416): text "Short address available"
rectangle at (95,430)-(246,451): text "Member of the group"
rounded rectangle at (140,80)-(676,116): text "DALI Line %s"; shows DALI_Config.bDali_Linie; tooltip You can change the DALI Line only on the home page.
rectangle at (85,250)-(116,281): text "17"; alarm colour if DALI_Config.Kurzadr[17]
rectangle at (85,250)-(116,281): text "17"; invisible if not DALI_Config.Kurzadr[17]; alarm colour if DALI_Config.Gruppenadr[17]; toggles DALI_Config.Gruppenadr[17]
rectangle at (125,250)-(156,281): text "18"; alarm colour if DALI_Config.Kurzadr[18]
rectangle at (125,250)-(156,281): text "18"; invisible if not DALI_Config.Kurzadr[18]; alarm colour if DALI_Config.Gruppenadr[18]; toggles DALI_Config.Gruppenadr[18]
rectangle at (165,250)-(196,281): text "19"; alarm colour if DALI_Config.Kurzadr[19]
rectangle at (165,250)-(196,281): text "19"; invisible if not DALI_Config.Kurzadr[19]; alarm colour if DALI_Config.Gruppenadr[19]; toggles DALI_Config.Gruppenadr[19]
rectangle at (205,250)-(236,281): text "20"; alarm colour if DALI_Config.Kurzadr[20]
rectangle at (205,250)-(236,281): text "20"; invisible if not DALI_Config.Kurzadr[20]; alarm colour if DALI_Config.Gruppenadr[20]; toggles DALI_Config.Gruppenadr[20]
rectangle at (245,250)-(276,281): text "21"; alarm colour if DALI_Config.Kurzadr[21]
rectangle at (245,250)-(276,281): text "21"; invisible if not DALI_Config.Kurzadr[21]; alarm colour if DALI_Config.Gruppenadr[21]; toggles DALI_Config.Gruppenadr[21]
rectangle at (285,250)-(316,281): text "22"; alarm colour if DALI_Config.Kurzadr[22]
rectangle at (285,250)-(316,281): text "22"; invisible if not DALI_Config.Kurzadr[22]; alarm colour if DALI_Config.Gruppenadr[22]; toggles DALI_Config.Gruppenadr[22]
rectangle at (325,250)-(356,281): text "23"; alarm colour if DALI_Config.Kurzadr[23]
rectangle at (325,250)-(356,281): text "23"; invisible if not DALI_Config.Kurzadr[23]; alarm colour if DALI_Config.Gruppenadr[23]; toggles DALI_Config.Gruppenadr[23]
rectangle at (365,250)-(396,281): text "24"; alarm colour if DALI_Config.Kurzadr[24]
rectangle at (365,250)-(396,281): text "24"; invisible if not DALI_Config.Kurzadr[24]; alarm colour if DALI_Config.Gruppenadr[24]; toggles DALI_Config.Gruppenadr[24]
rectangle at (405,250)-(436,281): text "25"; alarm colour if DALI_Config.Kurzadr[25]
rectangle at (405,250)-(436,281): text "25"; invisible if not DALI_Config.Kurzadr[25]; alarm colour if DALI_Config.Gruppenadr[25]; toggles DALI_Config.Gruppenadr[25]
rectangle at (445,250)-(476,281): text "26"; alarm colour if DALI_Config.Kurzadr[26]
rectangle at (445,250)-(476,281): text "26"; invisible if not DALI_Config.Kurzadr[26]; alarm colour if DALI_Config.Gruppenadr[26]; toggles DALI_Config.Gruppenadr[26]
rectangle at (485,250)-(516,281): text "27"; alarm colour if DALI_Config.Kurzadr[27]
rectangle at (485,250)-(516,281): text "27"; invisible if not DALI_Config.Kurzadr[27]; alarm colour if DALI_Config.Gruppenadr[27]; toggles DALI_Config.Gruppenadr[27]
rectangle at (525,250)-(556,281): text "28"; alarm colour if DALI_Config.Kurzadr[28]
rectangle at (525,250)-(556,281): text "28"; invisible if not DALI_Config.Kurzadr[28]; alarm colour if DALI_Config.Gruppenadr[28]; toggles DALI_Config.Gruppenadr[28]
rectangle at (565,250)-(596,281): text "29"; alarm colour if DALI_Config.Kurzadr[29]
rectangle at (565,250)-(596,281): text "29"; invisible if not DALI_Config.Kurzadr[29]; alarm colour if DALI_Config.Gruppenadr[29]; toggles DALI_Config.Gruppenadr[29]
rectangle at (605,250)-(636,281): text "30"; alarm colour if DALI_Config.Kurzadr[30]
rectangle at (605,250)-(636,281): text "30"; invisible if not DALI_Config.Kurzadr[30]; alarm colour if DALI_Config.Gruppenadr[30]; toggles DALI_Config.Gruppenadr[30]
rectangle at (645,250)-(676,281): text "31"; alarm colour if DALI_Config.Kurzadr[31]
rectangle at (645,250)-(676,281): text "31"; invisible if not DALI_Config.Kurzadr[31]; alarm colour if DALI_Config.Gruppenadr[31]; toggles DALI_Config.Gruppenadr[31]
rectangle at (685,250)-(716,281): text "32"; alarm colour if DALI_Config.Kurzadr[32]
rectangle at (685,250)-(716,281): text "32"; invisible if not DALI_Config.Kurzadr[32]; alarm colour if DALI_Config.Gruppenadr[32]; toggles DALI_Config.Gruppenadr[32]
rectangle at (85,290)-(116,321): text "33"; alarm colour if DALI_Config.Kurzadr[33]
rectangle at (85,290)-(116,321): text "33"; invisible if not DALI_Config.Kurzadr[33]; alarm colour if DALI_Config.Gruppenadr[33]; toggles DALI_Config.Gruppenadr[33]
rectangle at (125,290)-(156,321): text "34"; alarm colour if DALI_Config.Kurzadr[34]
rectangle at (125,290)-(156,321): text "34"; invisible if not DALI_Config.Kurzadr[34]; alarm colour if DALI_Config.Gruppenadr[34]; toggles DALI_Config.Gruppenadr[34]
rectangle at (165,290)-(196,321): text "35"; alarm colour if DALI_Config.Kurzadr[35]
rectangle at (165,290)-(196,321): text "35"; invisible if not DALI_Config.Kurzadr[35]; alarm colour if DALI_Config.Gruppenadr[35]; toggles DALI_Config.Gruppenadr[35]
rectangle at (205,290)-(236,321): text "36"; alarm colour if DALI_Config.Kurzadr[36]
rectangle at (205,290)-(236,321): text "36"; invisible if not DALI_Config.Kurzadr[36]; alarm colour if DALI_Config.Gruppenadr[36]; toggles DALI_Config.Gruppenadr[36]
rectangle at (245,290)-(276,321): text "37"; alarm colour if DALI_Config.Kurzadr[37]
rectangle at (245,290)-(276,321): text "37"; invisible if not DALI_Config.Kurzadr[37]; alarm colour if DALI_Config.Gruppenadr[37]; toggles DALI_Config.Gruppenadr[37]
rectangle at (285,290)-(316,321): text "38"; alarm colour if DALI_Config.Kurzadr[38]
rectangle at (285,290)-(316,321): text "38"; invisible if not DALI_Config.Kurzadr[38]; alarm colour if DALI_Config.Gruppenadr[38]; toggles DALI_Config.Gruppenadr[38]
rectangle at (325,290)-(356,321): text "39"; alarm colour if DALI_Config.Kurzadr[39]
rectangle at (325,290)-(356,321): text "39"; invisible if not DALI_Config.Kurzadr[39]; alarm colour if DALI_Config.Gruppenadr[39]; toggles DALI_Config.Gruppenadr[39]
rectangle at (365,290)-(396,321): text "40"; alarm colour if DALI_Config.Kurzadr[40]
rectangle at (365,290)-(396,321): text "40"; invisible if not DALI_Config.Kurzadr[40]; alarm colour if DALI_Config.Gruppenadr[40]; toggles DALI_Config.Gruppenadr[40]
rectangle at (405,290)-(436,321): text "41"; alarm colour if DALI_Config.Kurzadr[41]
rectangle at (405,290)-(436,321): text "41"; invisible if not DALI_Config.Kurzadr[41]; alarm colour if DALI_Config.Gruppenadr[41]; toggles DALI_Config.Gruppenadr[41]
rectangle at (445,290)-(476,321): text "42"; alarm colour if DALI_Config.Kurzadr[42]
rectangle at (445,290)-(476,321): text "42"; invisible if not DALI_Config.Kurzadr[42]; alarm colour if DALI_Config.Gruppenadr[42]; toggles DALI_Config.Gruppenadr[42]
rectangle at (485,290)-(516,321): text "43"; alarm colour if DALI_Config.Kurzadr[43]
rectangle at (485,290)-(516,321): text "43"; invisible if not DALI_Config.Kurzadr[43]; alarm colour if DALI_Config.Gruppenadr[43]; toggles DALI_Config.Gruppenadr[43]
rectangle at (525,290)-(556,321): text "44"; alarm colour if DALI_Config.Kurzadr[44]
rectangle at (525,290)-(556,321): text "44"; invisible if not DALI_Config.Kurzadr[44]; alarm colour if DALI_Config.Gruppenadr[44]; toggles DALI_Config.Gruppenadr[44]
rectangle at (565,290)-(596,321): text "45"; alarm colour if DALI_Config.Kurzadr[45]
rectangle at (565,290)-(596,321): text "45"; invisible if not DALI_Config.Kurzadr[45]; alarm colour if DALI_Config.Gruppenadr[45]; toggles DALI_Config.Gruppenadr[45]
rectangle at (605,290)-(636,321): text "46"; alarm colour if DALI_Config.Kurzadr[46]
rectangle at (605,290)-(636,321): text "46"; invisible if not DALI_Config.Kurzadr[46]; alarm colour if DALI_Config.Gruppenadr[46]; toggles DALI_Config.Gruppenadr[46]
rectangle at (645,290)-(676,321): text "47"; alarm colour if DALI_Config.Kurzadr[47]
rectangle at (645,290)-(676,321): text "47"; invisible if not DALI_Config.Kurzadr[47]; alarm colour if DALI_Config.Gruppenadr[47]; toggles DALI_Config.Gruppenadr[47]
rectangle at (685,290)-(716,321): text "48"; alarm colour if DALI_Config.Kurzadr[48]
rectangle at (685,290)-(716,321): text "48"; invisible if not DALI_Config.Kurzadr[48]; alarm colour if DALI_Config.Gruppenadr[48]; toggles DALI_Config.Gruppenadr[48]
rectangle at (85,330)-(116,361): text "49"; alarm colour if DALI_Config.Kurzadr[49]
rectangle at (85,330)-(116,361): text "49"; invisible if not DALI_Config.Kurzadr[49]; alarm colour if DALI_Config.Gruppenadr[49]; toggles DALI_Config.Gruppenadr[49]
rectangle at (125,330)-(156,361): text "50"; alarm colour if DALI_Config.Kurzadr[50]
rectangle at (125,330)-(156,361): text "50"; invisible if not DALI_Config.Kurzadr[50]; alarm colour if DALI_Config.Gruppenadr[50]; toggles DALI_Config.Gruppenadr[50]
rectangle at (165,330)-(196,361): text "51"; alarm colour if DALI_Config.Kurzadr[51]
rectangle at (165,330)-(196,361): text "51"; invisible if not DALI_Config.Kurzadr[51]; alarm colour if DALI_Config.Gruppenadr[51]; toggles DALI_Config.Gruppenadr[51]
rectangle at (205,330)-(236,361): text "52"; alarm colour if DALI_Config.Kurzadr[52]
rectangle at (205,330)-(236,361): text "52"; invisible if not DALI_Config.Kurzadr[52]; alarm colour if DALI_Config.Gruppenadr[52]; toggles DALI_Config.Gruppenadr[52]
rectangle at (245,330)-(276,361): text "53"; alarm colour if DALI_Config.Kurzadr[53]
rectangle at (245,330)-(276,361): text "53"; invisible if not DALI_Config.Kurzadr[53]; alarm colour if DALI_Config.Gruppenadr[53]; toggles DALI_Config.Gruppenadr[53]
rectangle at (285,330)-(316,361): text "54"; alarm colour if DALI_Config.Kurzadr[54]
rectangle at (285,330)-(316,361): text "54"; invisible if not DALI_Config.Kurzadr[54]; alarm colour if DALI_Config.Gruppenadr[54]; toggles DALI_Config.Gruppenadr[54]
rectangle at (325,330)-(356,361): text "55"; alarm colour if DALI_Config.Kurzadr[55]
rectangle at (325,330)-(356,361): text "55"; invisible if not DALI_Config.Kurzadr[55]; alarm colour if DALI_Config.Gruppenadr[55]; toggles DALI_Config.Gruppenadr[55]
rectangle at (365,330)-(396,361): text "56"; alarm colour if DALI_Config.Kurzadr[56]
rectangle at (365,330)-(396,361): text "56"; invisible if not DALI_Config.Kurzadr[56]; alarm colour if DALI_Config.Gruppenadr[56]; toggles DALI_Config.Gruppenadr[56]
rectangle at (405,330)-(436,361): text "57"; alarm colour if DALI_Config.Kurzadr[57]
rectangle at (405,330)-(436,361): text "57"; invisible if not DALI_Config.Kurzadr[57]; alarm colour if DALI_Config.Gruppenadr[57]; toggles DALI_Config.Gruppenadr[57]
rectangle at (445,330)-(476,361): text "58"; alarm colour if DALI_Config.Kurzadr[58]
rectangle at (445,330)-(476,361): text "58"; invisible if not DALI_Config.Kurzadr[58]; alarm colour if DALI_Config.Gruppenadr[58]; toggles DALI_Config.Gruppenadr[58]
rectangle at (485,330)-(516,361): text "59"; alarm colour if DALI_Config.Kurzadr[59]
rectangle at (485,330)-(516,361): text "59"; invisible if not DALI_Config.Kurzadr[59]; alarm colour if DALI_Config.Gruppenadr[59]; toggles DALI_Config.Gruppenadr[59]
rectangle at (525,330)-(556,361): text "60"; alarm colour if DALI_Config.Kurzadr[60]
rectangle at (525,330)-(556,361): text "60"; invisible if not DALI_Config.Kurzadr[60]; alarm colour if DALI_Config.Gruppenadr[60]; toggles DALI_Config.Gruppenadr[60]
rectangle at (565,330)-(596,361): text "61"; alarm colour if DALI_Config.Kurzadr[61]
rectangle at (565,330)-(596,361): text "61"; invisible if not DALI_Config.Kurzadr[61]; alarm colour if DALI_Config.Gruppenadr[61]; toggles DALI_Config.Gruppenadr[61]
rectangle at (605,330)-(636,361): text "62"; alarm colour if DALI_Config.Kurzadr[62]
rectangle at (605,330)-(636,361): text "62"; invisible if not DALI_Config.Kurzadr[62]; alarm colour if DALI_Config.Gruppenadr[62]; toggles DALI_Config.Gruppenadr[62]
rectangle at (645,330)-(676,361): text "63"; alarm colour if DALI_Config.Kurzadr[63]
rectangle at (645,330)-(676,361): text "63"; invisible if not DALI_Config.Kurzadr[63]; alarm colour if DALI_Config.Gruppenadr[63]; toggles DALI_Config.Gruppenadr[63]
rectangle at (685,330)-(716,361): text "64"; alarm colour if DALI_Config.Kurzadr[64]
rectangle at (685,330)-(716,361): text "64"; invisible if not DALI_Config.Kurzadr[64]; alarm colour if DALI_Config.Gruppenadr[64]; toggles DALI_Config.Gruppenadr[64]
rectangle at (580,395)-(696,431): text "Blink time [sek]"
button at (240,440)-(376,476): text "Central Off"; taps DALI_Config.Aus; tooltip If you click the button "Central Off", all lamps in the network will be switched off.
button at (240,395)-(376,431): text "Central On"; taps DALI_Config.Ein; tooltip If you click the button "Central On", all lamps in the network will be switched on.
rectangle at (700,395)-(736,431): text "%s"; shows DALI_Config.bBlinkzeit; tooltip Enter blink time (3 - 255 seconds); editable
rectangle at (42,88)-(763,482): text "Please wait!"; invisible if NOT DALI_Config.Unsichtbar
67 more shapes without text or variables
*)

(* Visualisation GroupSceneConfiguration
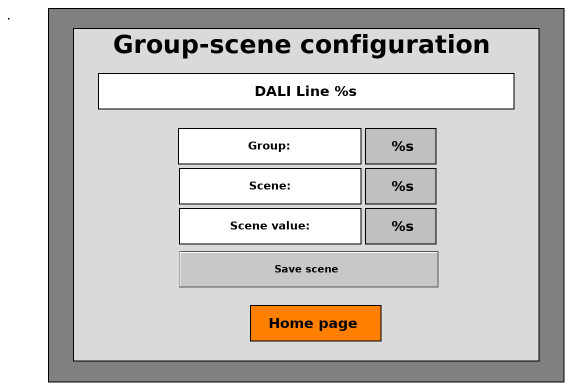
rectangle at (150,40)-(616,373): text "Group-scene configuration"
rounded rectangle at (327,317)-(458,353): text "Home page"; opens PLC_VISU; tooltip Back to home page
rounded rectangle at (175,85)-(591,121): text "DALI Line %s"; shows DALI_Config.bDali_Linie; tooltip You can change the DALI Line only on the home page.
rectangle at (255,140)-(438,176): text "Group:"
rectangle at (442,140)-(513,176): text "%s"; shows DALI_Config.sGroup; tooltip Enter the number of the group (1 - 16); editable
button at (256,263)-(515,299): text "Save scene"; taps DALI_Config.sSaveScene; tooltip Save the configured dim levels in the ECGs.
rectangle at (256,180)-(438,216): text "Scene:"
rectangle at (442,180)-(513,216): text "%s"; shows DALI_Config.sScene; tooltip Select scene 1 - 16; editable
rectangle at (256,220)-(438,256): text "Scene value:"
rectangle at (442,220)-(513,256): text "%s"; shows DALI_Config.sSceneValue; tooltip Select scene 1 - 16; editable
2 more shapes without text or variables
*)

